# B&R Automation Studio project TD52 (part 42)

#### c_anaCyclic.st - Zyklischer Code
```iecst
(*******************************************************************************
CUSTOMIZED: c_ana 		hardcoded customized analog inputs

This code is confidential and proprietary to the INNIO Company.
It may not be used in any form, or reproduced in any manner,
without written permission of the INNIO Company.
Copyright, INNIO Company, 2022

Customized modifications: -
------------------------

History:
-------
V3.90.0	??-??-2012  pankayrodney  	converted from LD
...
V4.01.0	13.11.2014 	zengerer		ADD AnalogIn Para.rCustAnaIn_LimLoLo[] and _HiHi[] and Alarm debug links
V4.02.0	24.06.2015 	zengerer		Cleanup, prototype entry[x] for documentation comments
V4.04.0 20-06-2016	Weitzer,		add CustAnaOut[17..50]
									add reserve controller output [41 .. 45]
V4.07.0 21.01.2019	zengerer		add some example lines in init to disable Reserve ANALOG IN Warning Signal Errors – NUMBER W1177 -
V4.07.1 09.05.2019	zengerer		add more bBlock[] example lines in init to disable Reserve ANALOG IN Warning Signal Errors W1336 - W1480
V4.11.1 31.01.2022	zengerer		new extended array ranges ONLY FOR USE WITH HMI Extension Package import!
V4.12.0 22.12.2022	zengerer		Outdated declarations removed: ParaFactoryDefault.bCustAnaIn_Set4mA[x], tUniAnaConf[x]
V4.13.0 21.09.2023	zengerer		Prepared spare analog output signal for VIS display (with unchanged scaling), constant for array declaration +check AO arrays

Instructions for use:
--------------------

AVOID HARDCODED Para.xxx VALUES!
You MAYBE want to enter SOME factory default values in the INIT section, but ONLY TO THE Para_FactoryDefault.xxx STRUCTURE!
._FactoryDefault values get read out only once at first controller startup, until the par_XX.dat files are automatically generated.
By this way the parameter values in Para.xxx would stay acessible according to XT4 parameter management process.

Outstandings:
------------

*******************************************************************************)

PROGRAM _CYCLIC

	(************************************************************)
	(*                                                          *)
	(*                   ANALOG INPUT SECTION                   *)
	(*                                                          *)
	(************************************************************)

//	(*Reserve analog input x *)									(* (CONFIGURATION EXAMPLE) *)
//	(*Reserveanalogwert x    *)									(* (KONFIGURATIONSBEISPIEL)*)
//	(*************************)
//	rReplaceMeWithLocaleVarName	:= IN_CU.tCustAnaIn[x].Ai;		(*edit according to project needs*) 														(*eigene Variable für Kundenanpassung hier anbinden*)
//	OUT_CU.rCustAnaIn[x] ;										(*Use this value for plant specific extensions in other metamodules (needs .vvm edit)*)		(*OUT- Modulschnittstelle zur möglichen Verwendung in anderer Module (.vvm editieren)*)
//
//	(*scaling parameter watch*)									(*scaling parameter are used in HAL only IF NO EPLAN SCALING DATA IS PROVIDED!	*)
//	Para.rCustAnaIn_ScalMin[x]	; 	MM2VIS.bMsg1177;			(* statement here is for watch info only. AVOID HARDCODED PARA VALUES *)
//	Para.rCustAnaIn_ScalMax[x]	;								(* statement here is for watch info only. AVOID HARDCODED PARA VALUES *)
//
//	(*warning and alarm limit watch*)
//	Para.rCustAnaIn_LimLoLo[x]	;	MM2VIS.bMsg8966;			(* Alarm HiHi and LoLo, statement here is for watch info only. AVOID HARDCODED PARA VALUES *)
//	Para.rCustAnaIn_LimLo[x]	;	MM2VIS.bMsg1301;			(* Warning, statement here is for watch info only. AVOID HARDCODED PARA VALUES *)
//	Para.rCustAnaIn_LimHi[x]	; 	MM2VIS.bMsg1302;			(* Warning, statement here is for watch info only. AVOID HARDCODED PARA VALUES *)
//	Para.rCustAnaIn_LimHiHi[x]	; 								(* 						statement here is for watch info only. AVOID HARDCODED PARA VALUES *)
//	Para.rCustAnaIn_Hy[x]	; 									(* 						statement here is for watch info only. AVOID HARDCODED PARA VALUES *)
//	Para.iCustAnaIn_MinMaxActive[x];							(* see task header for settings in Para File or in INIT Para_FactoryDefault.iCustAnaIn_MinMaxActive; statement here is for watch info only. *)
//  --> see also Documents - 'CustomizedSpareRegulars' for hints on repeatedly used customisations

	(*Reserve analog input 1 *)
	(*Reserveanalogwert 1    *)
	(*************************)
	rReplaceMeWithLocaleVarName	:= IN_CU.tCustAnaIn[1].Ai;		(*edit according to project needs*)
	OUT_CU.rCustAnaIn[1] ;

	(*scaling parameter watch*)
	Para.rCustAnaIn_ScalMin[1]	; 	MM2VIS.bMsg1177;
	Para.rCustAnaIn_ScalMax[1]	;
	(*warning and alarm limit watch*)
	Para.rCustAnaIn_LimHiHi[1]	; 	MM2VIS.bMsg8966;
	Para.rCustAnaIn_LimLo[1]	;	MM2VIS.bMsg1301;
	Para.rCustAnaIn_LimHi[1]	; 	MM2VIS.bMsg1302;
	Para.rCustAnaIn_LimLoLo[1]	;	MM2VIS.bMsg8966;
	Para.rCustAnaIn_Hy[1]	;
	Para.iCustAnaIn_MinMaxActive[1];

	(*Reserve analog input 2 *)
	(*Reserveanalogwert 2    *)
	(*************************)
	rReplaceMeWithLocaleVarName	:= IN_CU.tCustAnaIn[2].Ai;
	OUT_CU.rCustAnaIn[2] ;

	(*scaling parameter watch*)
	Para.rCustAnaIn_ScalMin[2]	;	MM2VIS.bMsg1178;
	Para.rCustAnaIn_ScalMax[2]	;
	(*warning and alarm limit watch*)
	Para.rCustAnaIn_LimHiHi[2]	; 	MM2VIS.bMsg8967;
	Para.rCustAnaIn_LimLo[2]	;	MM2VIS.bMsg1304;
	Para.rCustAnaIn_LimHi[2]	; 	MM2VIS.bMsg1305;
	Para.rCustAnaIn_LimLoLo[2]	;	MM2VIS.bMsg8967;
	Para.rCustAnaIn_Hy[2]	;
	Para.iCustAnaIn_MinMaxActive[2];

	(*Reserve analog input 3 *)
	(*Reserveanalogwert 3    *)
	(*************************)
	rReplaceMeWithLocaleVarName := IN_CU.tCustAnaIn[3].Ai;
	OUT_CU.rCustAnaIn[3] ;

	Para.rCustAnaIn_ScalMin[3]	;	MM2VIS.bMsg1179;
	Para.rCustAnaIn_ScalMax[3]	;
	(*warning and alarm limit watch*)
	Para.rCustAnaIn_LimLo[3]	;	MM2VIS.bMsg1307;
	Para.rCustAnaIn_LimHi[3]	; 	MM2VIS.bMsg1308;
	Para.rCustAnaIn_LimLoLo[3]	;	MM2VIS.bMsg8968;
	Para.rCustAnaIn_LimHiHi[3]	;
	Para.rCustAnaIn_Hy[3]	;
	Para.iCustAnaIn_MinMaxActive[3];

	(*Reserve analog input 4 *)
	(*Reserveanalogwert 4    *)
	(*************************)
	rReplaceMeWithLocaleVarName := IN_CU.tCustAnaIn[4].Ai;
	OUT_CU.rCustAnaIn[4] ;

	(*scaling parameter watch*)
	Para.rCustAnaIn_ScalMin[4]	;	 MM2VIS.bMsg1180;
	Para.rCustAnaIn_ScalMax[4]	;
	(*warning and alarm limit watch*)
	Para.rCustAnaIn_LimLo[4]	;	MM2VIS.bMsg1310;
	Para.rCustAnaIn_LimHi[4]	; 	MM2VIS.bMsg1311;
	Para.rCustAnaIn_LimLoLo[4]	;	MM2VIS.bMsg8969;
	Para.rCustAnaIn_LimHiHi[4]	;
	Para.rCustAnaIn_Hy[4]	;
	Para.iCustAnaIn_MinMaxActive[4];

	(*Reserve analog input 5 *)
	(*Reserveanalogwert 5    *)
	(*************************)
	rReplaceMeWithLocaleVarName := IN_CU.tCustAnaIn[5].Ai;
	OUT_CU.rCustAnaIn[5] ;

	(*scaling parameter watch*)
	Para.rCustAnaIn_ScalMin[5]	;	 MM2VIS.bMsg1181;
	Para.rCustAnaIn_ScalMax[5]	;
	(*warning and alarm limit watch*)
	Para.rCustAnaIn_LimLo[5]	;	MM2VIS.bMsg1313;
	Para.rCustAnaIn_LimHi[5]	; 	MM2VIS.bMsg1314;
	Para.rCustAnaIn_LimLoLo[5]	;	MM2VIS.bMsg8970;
	Para.rCustAnaIn_LimHiHi[5]	;

	(*Reserveanalogwert 6 *)
	(**********************)
	rReplaceMeWithLocaleVarName := IN_CU.tCustAnaIn[6].Ai;
	OUT_CU.rCustAnaIn[6] ;

	(*scaling parameter watch*)
	Para.rCustAnaIn_ScalMin[6]	;	 MM2VIS.bMsg1182;
	Para.rCustAnaIn_ScalMax[6]	;
	(*warning and alarm limit watch*)
	Para.rCustAnaIn_LimLo[6]	;	MM2VIS.bMsg1316;
	Para.rCustAnaIn_LimHi[6]	; 	MM2VIS.bMsg1317;
	Para.rCustAnaIn_LimLoLo[6]	;	MM2VIS.bMsg8971;
	Para.rCustAnaIn_LimHiHi[6]	;

	(*Reserveanalogwert 7 *)
	(**********************)
	rReplaceMeWithLocaleVarName := IN_CU.tCustAnaIn[7].Ai;
	OUT_CU.rCustAnaIn[7] ;

	(*scaling parameter watch*)
	Para.rCustAnaIn_ScalMin[7]	;	 MM2VIS.bMsg1183;
	Para.rCustAnaIn_ScalMax[7]	;
	(*warning and alarm limit watch*)
	Para.rCustAnaIn_LimLo[7]	;	MM2VIS.bMsg1319;
	Para.rCustAnaIn_LimHi[7]	; 	MM2VIS.bMsg1320;
	Para.rCustAnaIn_LimLoLo[7]	;	MM2VIS.bMsg8972;
	Para.rCustAnaIn_LimHiHi[7]	;

	(*Reserveanalogwert 8 *)
	(**********************)
	rReplaceMeWithLocaleVarName	:= IN_CU.tCustAnaIn[8].Ai;
	OUT_CU.rCustAnaIn[8] ;

	(*scaling parameter watch*)
	Para.rCustAnaIn_ScalMin[8]	;	 MM2VIS.bMsg1184;
	Para.rCustAnaIn_ScalMax[8]	;
	(*warning and alarm limit watch*)
	Para.rCustAnaIn_LimLo[8]	;	MM2VIS.bMsg1322;
	Para.rCustAnaIn_LimHi[8]	; 	MM2VIS.bMsg1323;
	Para.rCustAnaIn_LimLoLo[8]	;	MM2VIS.bMsg8973;
	Para.rCustAnaIn_LimHiHi[8]	;

	(*Reserveanalogwert 9 *)
	(**********************)
	rReplaceMeWithLocaleVarName	:= IN_CU.tCustAnaIn[9].Ai;
	OUT_CU.rCustAnaIn[9] := 0;
	MM2VIS.bMsg1327;

	(*scaling parameter watch*)
	Para.rCustAnaIn_ScalMin[9]	;	MM2VIS.bMsg1327;	(*!change in numbering pattern!*)
	Para.rCustAnaIn_ScalMax[9]	;
	(*warning and alarm limit watch*)
	Para.rCustAnaIn_LimLo[9]	;	MM2VIS.bMsg1325;
	Para.rCustAnaIn_LimHi[9]	; 	MM2VIS.bMsg1326;
	Para.rCustAnaIn_LimLoLo[9]	;	MM2VIS.bMsg8974;
	Para.rCustAnaIn_LimHiHi[9]	;

	(*Reserveanalogwert 10 *)
	(**********************)
	rReplaceMeWithLocaleVarName	:= IN_CU.tCustAnaIn[10].Ai;
	OUT_CU.rCustAnaIn[10] := 0;
	MM2VIS.bMsg1330;

	(*scaling parameter watch*)
	Para.rCustAnaIn_ScalMin[10]	;	MM2VIS.bMsg1330;
	Para.rCustAnaIn_ScalMax[10]	;
	(*warning and alarm limit watch*)
	Para.rCustAnaIn_LimLo[10]	;	MM2VIS.bMsg1328;
	Para.rCustAnaIn_LimHi[10]	; 	MM2VIS.bMsg1329;
	Para.rCustAnaIn_LimLoLo[10]	;	MM2VIS.bMsg8975;
	Para.rCustAnaIn_LimHiHi[10]	;
	Para.rCustAnaIn_Hy[10]	;
	Para.iCustAnaIn_MinMaxActive[10];

	(*Reserveanalogwert 11 *)
	(**********************)
	rReplaceMeWithLocaleVarName	:= IN_CU.tCustAnaIn[11].Ai;
	OUT_CU.rCustAnaIn[11] := 0;
	MM2VIS.bMsg1333;

	(*scaling parameter watch*)
	Para.rCustAnaIn_ScalMin[11]	;	MM2VIS.bMsg1333;
	Para.rCustAnaIn_ScalMax[11]	;
	(*warning and alarm limit watch*)
	Para.rCustAnaIn_LimLo[11]	;	MM2VIS.bMsg1331;
	Para.rCustAnaIn_LimHi[11]	; 	MM2VIS.bMsg1332;
	Para.rCustAnaIn_LimLoLo[11]	;	MM2VIS.bMsg8976;
	Para.rCustAnaIn_LimHiHi[11]	;

	(*Reserveanalogwert 12 *)
	(**********************)
	rReplaceMeWithLocaleVarName	:= IN_CU.tCustAnaIn[12].Ai;
	OUT_CU.rCustAnaIn[12] := 0;
	MM2VIS.bMsg1336;
	(*...*)

	(*Reserveanalogwert 13 *)
	(**********************)
	rReplaceMeWithLocaleVarName	:= IN_CU.tCustAnaIn[13].Ai;
	OUT_CU.rCustAnaIn[13] := 0;
	MM2VIS.bMsg1339;

	(*Reserveanalogwert 14 *)
	(**********************)
	rReplaceMeWithLocaleVarName := IN_CU.tCustAnaIn[14].Ai;
	OUT_CU.rCustAnaIn[14] := 0;
	MM2VIS.bMsg1342;

	(*Reserveanalogwert 15 *)
	(**********************)
	rReplaceMeWithLocaleVarName	:= IN_CU.tCustAnaIn[15].Ai;
	OUT_CU.rCustAnaIn[15] := 0;
	MM2VIS.bMsg1345;

	(*Reserveanalogwert 16 *)
	(**********************)
	rReplaceMeWithLocaleVarName	:= IN_CU.tCustAnaIn[16].Ai;
	OUT_CU.rCustAnaIn[16] := 0;
	MM2VIS.bMsg1348;

	(*Reserveanalogwert 17 *)
	(**********************)
	rReplaceMeWithLocaleVarName	:= IN_CU.tCustAnaIn[17].Ai;
	OUT_CU.rCustAnaIn[17] := 0;
	MM2VIS.bMsg1351;

	(*Reserveanalogwert 18 *)
	(**********************)
	rReplaceMeWithLocaleVarName	:= IN_CU.tCustAnaIn[18].Ai;
	OUT_CU.rCustAnaIn[18] := 0;
	MM2VIS.bMsg1354;

	(*Reserveanalogwert 19 *)
	(**********************)
	rReplaceMeWithLocaleVarName	:= IN_CU.tCustAnaIn[19].Ai;
	OUT_CU.rCustAnaIn[19] := 0;
	MM2VIS.bMsg1357;

	(*Reserveanalogwert 20 *)
	(**********************)
	rReplaceMeWithLocaleVarName	:= IN_CU.tCustAnaIn[20].Ai;
	OUT_CU.rCustAnaIn[20] := 0;

	(*scaling parameter watch*)
	Para.rCustAnaIn_ScalMin[20]	;	MM2VIS.bMsg1360;
	Para.rCustAnaIn_ScalMax[20]	;
	(*warning and alarm limit watch*)
	Para.rCustAnaIn_LimLo[20]	;	MM2VIS.bMsg1358;
	Para.rCustAnaIn_LimHi[20]	; 	MM2VIS.bMsg1359;
	Para.rCustAnaIn_LimLoLo[20]	;	MM2VIS.bMsg8985;
	Para.rCustAnaIn_LimHiHi[20]	;
	Para.rCustAnaIn_Hy[20]	;
	Para.iCustAnaIn_MinMaxActive[20];

	(*Reserveanalogwert 21 *)
	(**********************)
	rReplaceMeWithLocaleVarName	:= IN_CU.tCustAnaIn[21].Ai;
	OUT_CU.rCustAnaIn[21] := 0;

	(*scaling parameter watch*)
	Para.rCustAnaIn_ScalMin[21]	;	MM2VIS.bMsg1363;
	Para.rCustAnaIn_ScalMax[21]	;
	(*warning and alarm limit watch*)
	Para.rCustAnaIn_LimLo[21]	;	MM2VIS.bMsg1361;
	Para.rCustAnaIn_LimHi[21]	; 	MM2VIS.bMsg1362;
	Para.rCustAnaIn_LimLoLo[21]	;	MM2VIS.bMsg8986;
	Para.rCustAnaIn_LimHiHi[21]	;
	Para.rCustAnaIn_Hy[21]	;
	Para.iCustAnaIn_MinMaxActive[21];

	(*Reserveanalogwert 22 *)
	(**********************)
	rReplaceMeWithLocaleVarName	:= IN_CU.tCustAnaIn[22].Ai;
	OUT_CU.rCustAnaIn[22] := 0;
	MM2VIS.bMsg1366;

	(*Reserveanalogwert 23 *)
	(**********************)
	rReplaceMeWithLocaleVarName	:= IN_CU.tCustAnaIn[23].Ai;
	OUT_CU.rCustAnaIn[23] := 0;
	MM2VIS.bMsg1369;

	(*Reserveanalogwert 24 *)
	(**********************)
	rReplaceMeWithLocaleVarName	:= IN_CU.tCustAnaIn[24].Ai;
	OUT_CU.rCustAnaIn[24] := 0;

	(*Reserveanalogwert 25 *)
	(**********************)
	rReplaceMeWithLocaleVarName	:= IN_CU.tCustAnaIn[25].Ai;
	OUT_CU.rCustAnaIn[25] := 0;

	(*Reserveanalogwert 26 *)
	(**********************)
	rReplaceMeWithLocaleVarName	:= IN_CU.tCustAnaIn[26].Ai;
	OUT_CU.rCustAnaIn[26] := 0;

	(*Reserveanalogwert 27 *)
	(**********************)
	rReplaceMeWithLocaleVarName	:= IN_CU.tCustAnaIn[27].Ai;
	OUT_CU.rCustAnaIn[27] := 0;

	(*Reserveanalogwert 28 *)
	(**********************)
	rReplaceMeWithLocaleVarName	:= IN_CU.tCustAnaIn[28].Ai;
	OUT_CU.rCustAnaIn[28] := 0;

	(*Reserveanalogwert 29 *)
	(**********************)
	rReplaceMeWithLocaleVarName	:= IN_CU.tCustAnaIn[29].Ai;
	OUT_CU.rCustAnaIn[29] := 0;

	(*Reserve analog value  30 *)
	(**************************)
	rReplaceMeWithLocaleVarName	:= IN_CU.tCustAnaIn[30].Ai;
	OUT_CU.rCustAnaIn[30] := 0;

	(*scaling parameter watch*)
	Para.rCustAnaIn_ScalMin[30]	;	MM2VIS.bMsg1390;	 	(* ANALOG IN 30 Warning Signal Error. statement here is for watch info only. *)
	Para.rCustAnaIn_ScalMax[30]	;
	(*warning and alarm limit watch*)
	Para.rCustAnaIn_LimLo[30]	;	MM2VIS.bMsg1388;
	Para.rCustAnaIn_LimHi[30]	; 	MM2VIS.bMsg1389;
	Para.rCustAnaIn_LimLoLo[30]	;	MM2VIS.bMsg8995;
	Para.rCustAnaIn_LimHiHi[30]	;
	Para.rCustAnaIn_Hy[30]	;
	Para.iCustAnaIn_MinMaxActive[30];

	(*Reserve analog value  31 *)
	(**************************)
	rReplaceMeWithLocaleVarName	:= IN_CU.tCustAnaIn[31].Ai;
	OUT_CU.rCustAnaIn[31] := 0;

	(*scaling parameter watch*)
	Para.rCustAnaIn_ScalMin[31]	;	MM2VIS.bMsg1393;		(* ANALOG IN 31 Warning Signal Error. statement here is for watch info only. *)
	Para.rCustAnaIn_ScalMax[31]	;
	(*warning limit watch*)
	Para.rCustAnaIn_LimLo[31]	;	MM2VIS.bMsg1391;  		(* ANALOG IN 31 Warning Limit LOW,  statement here is for watch info only.   *)
	Para.rCustAnaIn_LimHi[31]	; 	MM2VIS.bMsg1392;  		(* ANALOG IN 31 Warning Limit HIGH, statement here is for watch info only.   *)
(*!*)Para.rCustAnaIn_LimLoLo[31];	MM2VIS.bMsg8998;		(*!	Collective Alarm for Analog inputs 31-60:  limit alarms LoLo ! *)	(* Statement here for watch info only *)
(*!*)Para.rCustAnaIn_LimHiHi[31];	MM2VIS.bMsg8999;		(*!	Collective Alarm for Analog inputs 31-60:  limit alarms HiHi  Statement here for watch info only *)
	Para.rCustAnaIn_Hy[31]	;
	Para.iCustAnaIn_MinMaxActive[31];

	(*Reserve analog value  32 *)
	(**************************)
	rReplaceMeWithLocaleVarName	:= IN_CU.tCustAnaIn[32].Ai;
	OUT_CU.rCustAnaIn[32] := 0;

	(*scaling parameter watch*)
	Para.rCustAnaIn_ScalMin[32]	;	MM2VIS.bMsg1396;		(* ANALOG IN 32 Warning Signal Error. statement here is for watch info only. *)
	Para.rCustAnaIn_ScalMax[32]	;
	(*warning and alarm limit watch*)
	Para.rCustAnaIn_LimLo[32]	;	MM2VIS.bMsg1394;  		(* ANALOG IN 32 Warning Limit LOW,  statement here is for watch info only.   *)
	Para.rCustAnaIn_LimHi[32]	; 	MM2VIS.bMsg1395;  		(* ANALOG IN 32 Warning Limit HIGH, statement here is for watch info only.   *)
	Para.rCustAnaIn_Hy[32]	;
	Para.iCustAnaIn_MinMaxActive[32];

	(*Reserve analog value  33 *)
	(**************************)
	rReplaceMeWithLocaleVarName	:= IN_CU.tCustAnaIn[33].Ai;
	OUT_CU.rCustAnaIn[33] := 0;

	(*scaling parameter watch*)
	Para.rCustAnaIn_ScalMin[33]	;	MM2VIS.bMsg1399;
	Para.rCustAnaIn_ScalMax[33]	;
	(*warning and alarm limit watch*)
	Para.rCustAnaIn_LimLo[33]	;	MM2VIS.bMsg1397;
	Para.rCustAnaIn_LimHi[33]	; 	MM2VIS.bMsg1398;
	Para.rCustAnaIn_Hy[33]	;
	Para.iCustAnaIn_MinMaxActive[33];

	(*Reserve analog value  34 *)
	(**************************)
	rReplaceMeWithLocaleVarName	:= IN_CU.tCustAnaIn[34].Ai;
	OUT_CU.rCustAnaIn[34] := 0;

	(*scaling parameter watch*)
	Para.rCustAnaIn_ScalMin[34]	;	MM2VIS.bMsg1402;
	Para.rCustAnaIn_ScalMax[34]	;
	(*warning and alarm limit watch*)
	Para.rCustAnaIn_LimLo[34]	;	MM2VIS.bMsg1400;
	Para.rCustAnaIn_LimHi[34]	; 	MM2VIS.bMsg1401;
	Para.rCustAnaIn_Hy[34]	;
	Para.iCustAnaIn_MinMaxActive[34];

	(*Reserve analog value  35 *)
	(**************************)
	rReplaceMeWithLocaleVarName	:= IN_CU.tCustAnaIn[35].Ai;
	OUT_CU.rCustAnaIn[35] := 0;

	(*scaling parameter watch*)
	Para.rCustAnaIn_ScalMin[35]	;	MM2VIS.bMsg1405;
	Para.rCustAnaIn_ScalMax[35]	;
	(*warning and alarm limit watch*)
	Para.rCustAnaIn_LimLo[35]	;	MM2VIS.bMsg1403;
	Para.rCustAnaIn_LimHi[35]	; 	MM2VIS.bMsg1404;
	Para.rCustAnaIn_Hy[35]	;
	Para.iCustAnaIn_MinMaxActive[35];

	(*Reserve analog value  36 *)
	(**************************)
	rReplaceMeWithLocaleVarName	:= IN_CU.tCustAnaIn[36].Ai;
	OUT_CU.rCustAnaIn[36] := 0;

	(*Reserve analog value  37 *)
	(**************************)
	rReplaceMeWithLocaleVarName	:= IN_CU.tCustAnaIn[37].Ai;
	OUT_CU.rCustAnaIn[37] := 0;

	(*Reserve analog value  38 *)
	(**************************)
	rReplaceMeWithLocaleVarName	:= IN_CU.tCustAnaIn[38].Ai;
	OUT_CU.rCustAnaIn[38] := 0;

	(*Reserve analog value  39 *)
	(**************************)
	rReplaceMeWithLocaleVarName	:= IN_CU.tCustAnaIn[39].Ai;
	OUT_CU.rCustAnaIn[39] := 0;

	(*Reserve analog value  40 *)
	(**************************)
	rReplaceMeWithLocaleVarName	:= IN_CU.tCustAnaIn[40].Ai;
	OUT_CU.rCustAnaIn[40] := 0;

	(*scaling parameter watch*)
	Para.rCustAnaIn_ScalMin[40]	;	MM2VIS.bMsg1420;		(* ANALOG IN 40 Warning Signal Error. statement here is for watch info only. *)
	Para.rCustAnaIn_ScalMax[40]	;
	(*warning and alarm limit watch*)
	Para.rCustAnaIn_LimLo[40]	;	MM2VIS.bMsg1418; 		(* ANALOG IN 40 Warning Limit LOW,  statement here is for watch info only.   *)
	Para.rCustAnaIn_LimHi[40]	; 	MM2VIS.bMsg1419; 		(* ANALOG IN 40 Warning Limit HIGH, statement here is for watch info only.   *)
	Para.rCustAnaIn_Hy[40]	;
	Para.iCustAnaIn_MinMaxActive[40];

	(*Reserve analog value  41 *)
	(**************************)
	rReplaceMeWithLocaleVarName	:= IN_CU.tCustAnaIn[41].Ai;
	OUT_CU.rCustAnaIn[41] := 0;

	(*scaling parameter watch*)
	Para.rCustAnaIn_ScalMin[41]	;	MM2VIS.bMsg1423;		(* ANALOG IN 41 Warning Signal Error. statement here is for watch info only. *)
	Para.rCustAnaIn_ScalMax[41]	;
	(*warning and alarm limit watch*)
	Para.rCustAnaIn_LimLo[41]	;	MM2VIS.bMsg1421; 		(* ANALOG IN 41 Warning Limit LOW,  statement here is for watch info only.   *)
	Para.rCustAnaIn_LimHi[41]	; 	MM2VIS.bMsg1422; 		(* ANALOG IN 41 Warning Limit HIGH, statement here is for watch info only.   *)
	Para.rCustAnaIn_Hy[41]	;
	Para.iCustAnaIn_MinMaxActive[41];

	(*Reserve analog value  42 *)
	(**************************)
	rReplaceMeWithLocaleVarName	:= IN_CU.tCustAnaIn[42].Ai;
	OUT_CU.rCustAnaIn[42] := 0;

	(*Reserve analog value  43 *)
	(**************************)
	rReplaceMeWithLocaleVarName	:= IN_CU.tCustAnaIn[43].Ai;
	OUT_CU.rCustAnaIn[43] := 0;

	(*Reserve analog value  44 *)
	(**************************)
	rReplaceMeWithLocaleVarName	:= IN_CU.tCustAnaIn[44].Ai;
	OUT_CU.rCustAnaIn[44] := 0;

	(*Reserve analog value  45 *)
	(**************************)
	rReplaceMeWithLocaleVarName	:= IN_CU.tCustAnaIn[45].Ai;
	OUT_CU.rCustAnaIn[45] := 0;

	(*Reserve analog value  46 *)
	(**************************)
	rReplaceMeWithLocaleVarName	:= IN_CU.tCustAnaIn[46].Ai;
	OUT_CU.rCustAnaIn[46] := 0;

	(*Reserve analog value  47 *)
	(**************************)
	rReplaceMeWithLocaleVarName	:= IN_CU.tCustAnaIn[47].Ai;
	OUT_CU.rCustAnaIn[47] := 0;

	(*Reserve analog value  48 *)
	(**************************)
	rReplaceMeWithLocaleVarName	:= IN_CU.tCustAnaIn[48].Ai;
	OUT_CU.rCustAnaIn[48] := 0;

	(*Reserve analog value  49 *)
	(**************************)
	rReplaceMeWithLocaleVarName	:= IN_CU.tCustAnaIn[49].Ai;
	OUT_CU.rCustAnaIn[49] := 0;

	(*Reserve analog value  50 *)
	(**************************)
	rReplaceMeWithLocaleVarName	:= IN_CU.tCustAnaIn[50].Ai;
	OUT_CU.rCustAnaIn[50] := 0;

	(*scaling parameter watch*)
	Para.rCustAnaIn_ScalMin[50]	;	MM2VIS.bMsg1450;		(* ANALOG IN 50 Warning Signal Error. statement here is for watch info only. *)
	Para.rCustAnaIn_ScalMax[50]	;
	(*warning and alarm limit watch*)
	Para.rCustAnaIn_LimLo[50]	;	MM2VIS.bMsg1448;			(* ANALOG IN 50 Warning Limit LOW,  statement here is for watch info only.   *)
	Para.rCustAnaIn_LimHi[50]	; 	MM2VIS.bMsg1449;			(* ANALOG IN 50 Warning Limit HIGH, statement here is for watch info only.   *)
	Para.rCustAnaIn_Hy[50]	;
	Para.iCustAnaIn_MinMaxActive[50];

	(*Reserve analog value  51 *)
	(**************************)
	rReplaceMeWithLocaleVarName	:= IN_CU.tCustAnaIn[51].Ai;
	OUT_CU.rCustAnaIn[51] := 0;

	(*Reserve analog value  52 *)
	(**************************)
	rReplaceMeWithLocaleVarName	:= IN_CU.tCustAnaIn[52].Ai;
	OUT_CU.rCustAnaIn[52] := 0;

	(*Reserve analog value  53 *)
	(**************************)
	rReplaceMeWithLocaleVarName	:= IN_CU.tCustAnaIn[53].Ai;
	OUT_CU.rCustAnaIn[53] := 0;

	(*Reserve analog value  54 *)
	(**************************)
	rReplaceMeWithLocaleVarName	:= IN_CU.tCustAnaIn[54].Ai;
	OUT_CU.rCustAnaIn[54] := 0;

	(*Reserve analog value  55 *)
	(**************************)
	rReplaceMeWithLocaleVarName	:= IN_CU.tCustAnaIn[55].Ai;
	OUT_CU.rCustAnaIn[55] := 0;

	(*Reserve analog value  56 *)
	(**************************)
	rReplaceMeWithLocaleVarName	:= IN_CU.tCustAnaIn[56].Ai;
	OUT_CU.rCustAnaIn[56] := 0;

	(*Reserve analog value  57 *)
	(**************************)
	rReplaceMeWithLocaleVarName	:= IN_CU.tCustAnaIn[57].Ai;
	OUT_CU.rCustAnaIn[57] := 0;

	(*Reserve analog value  58 *)
	(**************************)
	rReplaceMeWithLocaleVarName	:= IN_CU.tCustAnaIn[58].Ai;
	OUT_CU.rCustAnaIn[58] := 0;

	(*Reserve analog value  59 *)
	(**************************)
	rReplaceMeWithLocaleVarName	:= IN_CU.tCustAnaIn[59].Ai;
	OUT_CU.rCustAnaIn[59] := 0;

	(*Reserve analog value 60 *)
	(**************************)
	rReplaceMeWithLocaleVarName	:= IN_CU.tCustAnaIn[60].Ai;
	OUT_CU.rCustAnaIn[60] := 0;

	(*scaling parameter watch*)
	Para.rCustAnaIn_ScalMin[60]	;	MM2VIS.bMsg1480;		(* ANALOG IN 60 Warning Signal Error. statement here is for watch info only. *)
	Para.rCustAnaIn_ScalMax[60]	;
	(*warning and alarm limit watch*)
	Para.rCustAnaIn_LimLo[60]	;MM2VIS.bMsg1478 ;			(* ANALOG IN 60 Warning Limit LOW,  statement here is for watch info only.   *)
	Para.rCustAnaIn_LimHi[60]	;MM2VIS.bMsg1479 ;			(* ANALOG IN 60 Warning Limit HIGH, statement here is for watch info only.   *)
	Para.rCustAnaIn_Hy[60]	;
	Para.iCustAnaIn_MinMaxActive[60];

	(********************************************************************************************************************************************)
	(* Reserve analog input 61 and above are not prepared in HMI default! - FOR USE ONLY WITH `HMI_Extension` Package! *)
	(* Analog inputs 61- and above have no alarm messages and HMI display prepared in default and need HMI_Update packets imported for function! *)
	(*********************************************************************************************************************************************)
	(*Reserve analog value  61 *)
	(**************************)
	rReplaceMeWithLocaleVarName	:= IN_CU.tCustAnaIn[61].Ai;
	OUT_CU.rCustAnaIn[61] := 0;

	(*Reserve analog value  62 *)
	(**************************)
	rReplaceMeWithLocaleVarName	:= IN_CU.tCustAnaIn[62].Ai;
	OUT_CU.rCustAnaIn[62] := 0;

	(*Reserve analog value  63 *)
	(**************************)
	rReplaceMeWithLocaleVarName	:= IN_CU.tCustAnaIn[63].Ai;
	OUT_CU.rCustAnaIn[63] := 0;

	(*Reserve analog value  64 *)
	(**************************)
	rReplaceMeWithLocaleVarName	:= IN_CU.tCustAnaIn[64].Ai;
	OUT_CU.rCustAnaIn[64] := 0;

	(*Reserve analog value  66 *)
	(**************************)
	rReplaceMeWithLocaleVarName	:= IN_CU.tCustAnaIn[65].Ai;
	OUT_CU.rCustAnaIn[65] := 0;

	(*Reserve analog value  66 *)
	(**************************)
	rReplaceMeWithLocaleVarName	:= IN_CU.tCustAnaIn[66].Ai;
	OUT_CU.rCustAnaIn[66] := 0;

	(*Reserve analog value  67 *)
	(**************************)
	rReplaceMeWithLocaleVarName	:= IN_CU.tCustAnaIn[67].Ai;
	OUT_CU.rCustAnaIn[67] := 0;

	(*Reserve analog value  68 *)
	(**************************)
	rReplaceMeWithLocaleVarName	:= IN_CU.tCustAnaIn[68].Ai;
	OUT_CU.rCustAnaIn[68] := 0;

	(*Reserve analog value  69 *)
	(**************************)
	rReplaceMeWithLocaleVarName	:= IN_CU.tCustAnaIn[69].Ai;
	OUT_CU.rCustAnaIn[69] := 0;

	(*Reserve analog value 70 *)
	(**************************)
	rReplaceMeWithLocaleVarName	:= IN_CU.tCustAnaIn[70].Ai;
	OUT_CU.rCustAnaIn[70] := 0;

	(*scaling parameter watch*)
	Para.rCustAnaIn_ScalMin[70]	;	MM2VIS.bMsg3810;		(* ANALOG IN 70 Warning Signal Error. statement here is for watch info only. *)
	Para.rCustAnaIn_ScalMax[70]	;
	(*warning and alarm limit watch*)
	Para.rCustAnaIn_LimLo[70]	;MM2VIS.bMsg3808 ;			(* ANALOG IN 70 Warning Limit LOW,  statement here is for watch info only.   *)
	Para.rCustAnaIn_LimHi[70]	;MM2VIS.bMsg3809 ;			(* ANALOG IN 70 Warning Limit HIGH, statement here is for watch info only.   *)
	Para.rCustAnaIn_Hy[70]	;
	Para.iCustAnaIn_MinMaxActive[70];

	(*Reserve analog value  71 *)
	(**************************)
	rReplaceMeWithLocaleVarName	:= IN_CU.tCustAnaIn[71].Ai;
	OUT_CU.rCustAnaIn[71] := 0;

	(*Reserve analog value  72 *)
	(**************************)
	rReplaceMeWithLocaleVarName	:= IN_CU.tCustAnaIn[72].Ai;
	OUT_CU.rCustAnaIn[72] := 0;

	(*Reserve analog value  73 *)
	(**************************)
	rReplaceMeWithLocaleVarName	:= IN_CU.tCustAnaIn[73].Ai;
	OUT_CU.rCustAnaIn[73] := 0;

	(*Reserve analog value  74 *)
	(**************************)
	rReplaceMeWithLocaleVarName	:= IN_CU.tCustAnaIn[74].Ai;
	OUT_CU.rCustAnaIn[74] := 0;

	(*Reserve analog value  75 *)
	(**************************)
	rReplaceMeWithLocaleVarName	:= IN_CU.tCustAnaIn[75].Ai;
	OUT_CU.rCustAnaIn[75] := 0;

	(*Reserve analog value  76 *)
	(**************************)
	rReplaceMeWithLocaleVarName	:= IN_CU.tCustAnaIn[76].Ai;
	OUT_CU.rCustAnaIn[76] := 0;

	(*Reserve analog value  77 *)
	(**************************)
	rReplaceMeWithLocaleVarName	:= IN_CU.tCustAnaIn[77].Ai;
	OUT_CU.rCustAnaIn[77] := 0;

	(*Reserve analog value  78 *)
	(**************************)
	rReplaceMeWithLocaleVarName	:= IN_CU.tCustAnaIn[78].Ai;
	OUT_CU.rCustAnaIn[78] := 0;

	(*Reserve analog value  79 *)
	(**************************)
	rReplaceMeWithLocaleVarName	:= IN_CU.tCustAnaIn[79].Ai;
	OUT_CU.rCustAnaIn[79] := 0;

	(*Reserve analog value 80 *)
	(**************************)
	rReplaceMeWithLocaleVarName	:= IN_CU.tCustAnaIn[80].Ai;
	OUT_CU.rCustAnaIn[80] := 0;

	(*scaling parameter watch*)
	Para.rCustAnaIn_ScalMin[80]	;	MM2VIS.bMsg3840;		(* ANALOG IN 80 Warning Signal Error. statement here is for watch info only. *)
	Para.rCustAnaIn_ScalMax[80]	;
	(*warning and alarm limit watch*)
	Para.rCustAnaIn_LimLo[80]	;MM2VIS.bMsg3838 ;			(* ANALOG IN 80 Warning Limit LOW,  statement here is for watch info only.   *)
	Para.rCustAnaIn_LimHi[80]	;MM2VIS.bMsg3839 ;			(* ANALOG IN 80 Warning Limit HIGH, statement here is for watch info only.   *)
	Para.rCustAnaIn_Hy[80]	;
	Para.iCustAnaIn_MinMaxActive[80];

	(*Reserve analog value  81 *)
	(**************************)
	rReplaceMeWithLocaleVarName	:= IN_CU.tCustAnaIn[81].Ai;
	OUT_CU.rCustAnaIn[81] := 0;

	(*Reserve analog value  82 *)
	(**************************)
	rReplaceMeWithLocaleVarName	:= IN_CU.tCustAnaIn[82].Ai;
	OUT_CU.rCustAnaIn[82] := 0;

	(*Reserve analog value  83 *)
	(**************************)
	rReplaceMeWithLocaleVarName	:= IN_CU.tCustAnaIn[83].Ai;
	OUT_CU.rCustAnaIn[83] := 0;

	(*Reserve analog value  84 *)
	(**************************)
	rReplaceMeWithLocaleVarName	:= IN_CU.tCustAnaIn[84].Ai;
	OUT_CU.rCustAnaIn[84] := 0;

	(*Reserve analog value  85 *)
	(**************************)
	rReplaceMeWithLocaleVarName	:= IN_CU.tCustAnaIn[85].Ai;
	OUT_CU.rCustAnaIn[85] := 0;

	(*Reserve analog value  86 *)
	(**************************)
	rReplaceMeWithLocaleVarName	:= IN_CU.tCustAnaIn[86].Ai;
	OUT_CU.rCustAnaIn[86] := 0;

	(*Reserve analog value  87 *)
	(**************************)
	rReplaceMeWithLocaleVarName	:= IN_CU.tCustAnaIn[87].Ai;
	OUT_CU.rCustAnaIn[87] := 0;

	(*Reserve analog value  88 *)
	(**************************)
	rReplaceMeWithLocaleVarName	:= IN_CU.tCustAnaIn[88].Ai;
	OUT_CU.rCustAnaIn[88] := 0;

	(*Reserve analog value  89 *)
	(**************************)
	rReplaceMeWithLocaleVarName	:= IN_CU.tCustAnaIn[89].Ai;
	OUT_CU.rCustAnaIn[89] := 0;

	(*Reserve analog value 90 *)
	(**************************)
	rReplaceMeWithLocaleVarName	:= IN_CU.tCustAnaIn[90].Ai;
	OUT_CU.rCustAnaIn[90] := 0;

	(*scaling parameter watch*)
	Para.rCustAnaIn_ScalMin[90]	;	MM2VIS.bMsg3870;		(* ANALOG IN 90 Warning Signal Error. statement here is for watch info only. *)
	Para.rCustAnaIn_ScalMax[90]	;
	(*warning and alarm limit watch*)
	Para.rCustAnaIn_LimLo[90]	;MM2VIS.bMsg3868 ;			(* ANALOG IN 90 Warning Limit LOW,  statement here is for watch info only.   *)
	Para.rCustAnaIn_LimHi[90]	;MM2VIS.bMsg3869 ;			(* ANALOG IN 90 Warning Limit HIGH, statement here is for watch info only.   *)
	Para.rCustAnaIn_Hy[90]	;
	Para.iCustAnaIn_MinMaxActive[90];

	(*Reserve analog value  91 *)
	(**************************)
	rReplaceMeWithLocaleVarName	:= IN_CU.tCustAnaIn[91].Ai;
	OUT_CU.rCustAnaIn[91] := 0;

	(*Reserve analog value  92 *)
	(**************************)
	rReplaceMeWithLocaleVarName	:= IN_CU.tCustAnaIn[92].Ai;
	OUT_CU.rCustAnaIn[92] := 0;

	(*Reserve analog value  93 *)
	(**************************)
	rReplaceMeWithLocaleVarName	:= IN_CU.tCustAnaIn[93].Ai;
	OUT_CU.rCustAnaIn[93] := 0;

	(*Reserve analog value  94 *)
	(**************************)
	rReplaceMeWithLocaleVarName	:= IN_CU.tCustAnaIn[94].Ai;
	OUT_CU.rCustAnaIn[94] := 0;

	(*Reserve analog value  95 *)
	(**************************)
	rReplaceMeWithLocaleVarName	:= IN_CU.tCustAnaIn[95].Ai;
	OUT_CU.rCustAnaIn[95] := 0;

	(*Reserve analog value  96 *)
	(**************************)
	rReplaceMeWithLocaleVarName	:= IN_CU.tCustAnaIn[96].Ai;
	OUT_CU.rCustAnaIn[96] := 0;

	(*Reserve analog value  97 *)
	(**************************)
	rReplaceMeWithLocaleVarName	:= IN_CU.tCustAnaIn[97].Ai;
	OUT_CU.rCustAnaIn[97] := 0;

	(*Reserve analog value  98 *)
	(**************************)
	rReplaceMeWithLocaleVarName	:= IN_CU.tCustAnaIn[98].Ai;
	OUT_CU.rCustAnaIn[98] := 0;

	(*Reserve analog value  99 *)
	(**************************)
	rReplaceMeWithLocaleVarName	:= IN_CU.tCustAnaIn[99].Ai;
	OUT_CU.rCustAnaIn[99] := 0;

	(*Reserve analog value 100 *)
	(**************************)
	rReplaceMeWithLocaleVarName	:= IN_CU.tCustAnaIn[100].Ai;
	OUT_CU.rCustAnaIn[100] := 0;

	(*scaling parameter watch*)
	Para.rCustAnaIn_ScalMin[100];	MM2VIS.bMsg3900;		(* ANALOG IN 100 Warning Signal Error. statement here is for watch info only. *)
	Para.rCustAnaIn_ScalMax[100];
	(*warning and alarm limit watch*)
	Para.rCustAnaIn_LimLo[100]	;MM2VIS.bMsg3898 ;			(* ANALOG IN 100 Warning Limit LOW,  statement here is for watch info only.   *)
	Para.rCustAnaIn_LimHi[100]	;MM2VIS.bMsg3899 ;			(* ANALOG IN 100 Warning Limit HIGH, statement here is for watch info only.   *)
	Para.rCustAnaIn_Hy[100]	;
	Para.iCustAnaIn_MinMaxActive[100];

	(*Reserve analog value  101 *)
	(**************************)
	rReplaceMeWithLocaleVarName	:= IN_CU.tCustAnaIn[101].Ai;
	OUT_CU.rCustAnaIn[101] := 0;

	(*Reserve analog value  102 *)
	(**************************)
	rReplaceMeWithLocaleVarName	:= IN_CU.tCustAnaIn[102].Ai;
	OUT_CU.rCustAnaIn[102] := 0;

	(*Reserve analog value  103 *)
	(**************************)
	rReplaceMeWithLocaleVarName	:= IN_CU.tCustAnaIn[103].Ai;
	OUT_CU.rCustAnaIn[103] := 0;

	(*Reserve analog value  104 *)
	(**************************)
	rReplaceMeWithLocaleVarName	:= IN_CU.tCustAnaIn[104].Ai;
	OUT_CU.rCustAnaIn[104] := 0;

	(*Reserve analog value  105 *)
	(**************************)
	rReplaceMeWithLocaleVarName	:= IN_CU.tCustAnaIn[105].Ai;
	OUT_CU.rCustAnaIn[105] := 0;

	(*Reserve analog value  106 *)
	(**************************)
	rReplaceMeWithLocaleVarName	:= IN_CU.tCustAnaIn[106].Ai;
	OUT_CU.rCustAnaIn[106] := 0;

	(*Reserve analog value  107 *)
	(**************************)
	rReplaceMeWithLocaleVarName	:= IN_CU.tCustAnaIn[107].Ai;
	OUT_CU.rCustAnaIn[107] := 0;

	(*Reserve analog value  108 *)
	(**************************)
	rReplaceMeWithLocaleVarName	:= IN_CU.tCustAnaIn[108].Ai;
	OUT_CU.rCustAnaIn[108] := 0;

	(*Reserve analog value  109 *)
	(**************************)
	rReplaceMeWithLocaleVarName	:= IN_CU.tCustAnaIn[109].Ai;
	OUT_CU.rCustAnaIn[109] := 0;

	(*Reserve analog value 110 *)
	(**************************)
	rReplaceMeWithLocaleVarName	:= IN_CU.tCustAnaIn[110].Ai;
	OUT_CU.rCustAnaIn[110] := 0;

	(*scaling parameter watch*)
	Para.rCustAnaIn_ScalMin[110];	MM2VIS.bMsg3930;		(* ANALOG IN 110 Warning Signal Error. statement here is for watch info only. *)
	Para.rCustAnaIn_ScalMax[110];
	(*warning and alarm limit watch*)
	Para.rCustAnaIn_LimLo[110]	;MM2VIS.bMsg3928 ;			(* ANALOG IN 110 Warning Limit LOW,  statement here is for watch info only.   *)
	Para.rCustAnaIn_LimHi[110]	;MM2VIS.bMsg3929 ;			(* ANALOG IN 110 Warning Limit HIGH, statement here is for watch info only.   *)
	Para.rCustAnaIn_Hy[110]	;
	Para.iCustAnaIn_MinMaxActive[110];

	(*Reserve analog value  111 *)
	(**************************)
	rReplaceMeWithLocaleVarName	:= IN_CU.tCustAnaIn[111].Ai;
	OUT_CU.rCustAnaIn[111] := 0;

	(*Reserve analog value  112 *)
	(**************************)
	rReplaceMeWithLocaleVarName	:= IN_CU.tCustAnaIn[112].Ai;
	OUT_CU.rCustAnaIn[112] := 0;

	(*Reserve analog value  113 *)
	(**************************)
	rReplaceMeWithLocaleVarName	:= IN_CU.tCustAnaIn[113].Ai;
	OUT_CU.rCustAnaIn[113] := 0;

	(*Reserve analog value  114 *)
	(**************************)
	rReplaceMeWithLocaleVarName	:= IN_CU.tCustAnaIn[114].Ai;
	OUT_CU.rCustAnaIn[114] := 0;

	(*Reserve analog value  115 *)
	(**************************)
	rReplaceMeWithLocaleVarName	:= IN_CU.tCustAnaIn[115].Ai;
	OUT_CU.rCustAnaIn[115] := 0;

	(*Reserve analog value  116 *)
	(**************************)
	rReplaceMeWithLocaleVarName	:= IN_CU.tCustAnaIn[116].Ai;
	OUT_CU.rCustAnaIn[116] := 0;

	(*Reserve analog value  117 *)
	(**************************)
	rReplaceMeWithLocaleVarName	:= IN_CU.tCustAnaIn[117].Ai;
	OUT_CU.rCustAnaIn[117] := 0;

	(*Reserve analog value  118 *)
	(**************************)
	rReplaceMeWithLocaleVarName	:= IN_CU.tCustAnaIn[118].Ai;
	OUT_CU.rCustAnaIn[118] := 0;

	(*Reserve analog value  119 *)
	(**************************)
	rReplaceMeWithLocaleVarName	:= IN_CU.tCustAnaIn[119].Ai;
	OUT_CU.rCustAnaIn[119] := 0;

	(*Reserve analog value 120 *)
	(**************************)
	rReplaceMeWithLocaleVarName	:= IN_CU.tCustAnaIn[120].Ai;
	OUT_CU.rCustAnaIn[120] := 0;

	(*scaling parameter watch*)
	Para.rCustAnaIn_ScalMin[120];	MM2VIS.bMsg3960;		(* ANALOG IN 120 Warning Signal Error. statement here is for watch info only. *)
	Para.rCustAnaIn_ScalMax[120];
	(*warning and alarm limit watch*)
	Para.rCustAnaIn_LimLo[120];		MM2VIS.bMsg3958 ;			(* ANALOG IN 120 Warning Limit LOW,  statement here is for watch info only.   *)
	Para.rCustAnaIn_LimHi[120];		MM2VIS.bMsg3959 ;			(* ANALOG IN 120 Warning Limit HIGH, statement here is for watch info only.   *)
	Para.rCustAnaIn_Hy[120];
	Para.iCustAnaIn_MinMaxActive[120];

	(*********************************************************************************************************************************)

	(*********************************************************************************************************************************)

	(********************************************************)
	(*                                                      *)
	(*                 ANALOG OUTPUT SECTION                *)
	(*                                                      *)
	(********************************************************)

//	(***************************)
//	(* Reserve analog output x *)								(* (CONFIGURATION EXAMPLE) *)
//	(* Reserveanalogausgang x  *)								(* (KONFIGURATIONSBEISPIEL)*)
//	(***************************)
//	OUT_CU.tCustAnaOut[x].Ao	:= rConnectYourVariableHere ;	(*eigene Variable für Kundenanpassung hier anbeinden*)	(*edit according to project needs*)
//
//	(*scaling parameter watch*)									(* scaling parameter are used in HAL only IF NO EPLAN SCALING DATA IS PROVIDED!	*)
//	Para.rCustAnaOut_ScalMin[x]	; 								(*[Customer Unit] 'software side' of scaling;	statement here is for watch info only. AVOID HARDCODED PARA VALUES *)
//	Para.rCustAnaOut_ScalMax[x]	;								(*[Customer Unit] 'software side' of scaling;	statement here is for watch info only. AVOID HARDCODED PARA VALUES *)
//	Para.rI_CustAnaOut_ScalMin[x] ; 	(* := 4; *)				(*[mA] 'hardware side' of scaling;				statement here is for watch info only. AVOID HARDCODED PARA VALUES *)
//	Para.rI_CustAnaOut_ScalMin[x] ;		(* := 20; *)			(*[mA] 'hardware side' of scaling;				statement here is for watch info only. AVOID HARDCODED PARA VALUES *)

	(* reserve analog output 1 *)
	OUT_CU.tCustAnaOut[1].Ao	:= rConnectYourVariableHere ;	(* change customized *)
	(*scaling parameter watch*)
	Para.rCustAnaOut_ScalMin[1]	;
	Para.rCustAnaOut_ScalMax[1]	;
	Para.rI_CustAnaOut_ScalMin[1] ;
	Para.rI_CustAnaOut_ScalMax[1] ;
	MM2VIS.rCustAnaOut[1] ; 								(*Example call of prepared spare analog output for VIS service display; OLD: MM2VIS.rCustAnaOut_Norm[1]  *)

	(* reserve analog output 2 *)
	OUT_CU.tCustAnaOut[2].Ao	:= rConnectYourVariableHere ;
	(*scaling parameter watch*)
	Para.rCustAnaOut_ScalMin[2]	;
	Para.rCustAnaOut_ScalMax[2]	;
	Para.rI_CustAnaOut_ScalMin[2] ;
	Para.rI_CustAnaOut_ScalMax[2] ;

	(* reserve analog output 3 *)
	OUT_CU.tCustAnaOut[3].Ao	:= rConnectYourVariableHere ;
	(*scaling parameter watch*)
	Para.rCustAnaOut_ScalMin[3]	;
	Para.rCustAnaOut_ScalMax[3]	;
	Para.rI_CustAnaOut_ScalMin[3] ;
	Para.rI_CustAnaOut_ScalMax[3] ;

	(* reserve analog output 4 *)
	OUT_CU.tCustAnaOut[4].Ao	:= rConnectYourVariableHere ;
	(*scaling parameter watch*)
	Para.rCustAnaOut_ScalMin[4]	;
	Para.rCustAnaOut_ScalMax[4]	;
	Para.rI_CustAnaOut_ScalMin[4] ;
	Para.rI_CustAnaOut_ScalMax[4] ;

	(* reserve analog output 5 *)
//	OUT_CU.tCustAnaOut[5].Ao	:= rConnectYourVariableHere ;	 	(*VSofti*)
	(*scaling parameter watch*)
	Para.rCustAnaOut_ScalMin[5]	;
	Para.rCustAnaOut_ScalMax[5]	;
	Para.rI_CustAnaOut_ScalMin[5] ;
	Para.rI_CustAnaOut_ScalMax[5] ;

	(* reserve analog output 6 *)
	OUT_CU.tCustAnaOut[6].Ao	:= rConnectYourVariableHere ;
	(*scaling parameter watch*)
	Para.rCustAnaOut_ScalMin[6]	;
	Para.rCustAnaOut_ScalMax[6]	;
	Para.rI_CustAnaOut_ScalMin[6] ;
	Para.rI_CustAnaOut_ScalMax[6] ;

	(* reserve analog output 7 *)
//	OUT_CU.tCustAnaOut[7].Ao	:= rConnectYourVariableHere ;	 	(*VSofti*)
	(*scaling parameter watch*)
	Para.rCustAnaOut_ScalMin[7]	;
	Para.rCustAnaOut_ScalMax[7]	;
	Para.rI_CustAnaOut_ScalMin[7] ;
	Para.rI_CustAnaOut_ScalMax[7] ;

	(* reserve analog output 8 *)
//	OUT_CU.tCustAnaOut[8].Ao	:= rConnectYourVariableHere ;	 	(*VSofti*)
	(*scaling parameter watch*)
	Para.rCustAnaOut_ScalMin[8]	;
	Para.rCustAnaOut_ScalMax[8]	;
	Para.rI_CustAnaOut_ScalMin[8] ;
	Para.rI_CustAnaOut_ScalMax[8] ;

	(* reserve analog output 9 *)
//	OUT_CU.tCustAnaOut[9].Ao	:= rConnectYourVariableHere ;	 	(*VSofti*)
	(*scaling parameter watch*)
	Para.rCustAnaOut_ScalMin[9]	;
	Para.rCustAnaOut_ScalMax[9]	;
	Para.rI_CustAnaOut_ScalMin[9] ;
	Para.rI_CustAnaOut_ScalMax[9] ;

	(* reserve analog output 10 *)
//	OUT_CU.tCustAnaOut[10].Ao	:= rConnectYourVariableHere ;	 	(*VSofti*)
	(*scaling parameter watch*)
	Para.rCustAnaOut_ScalMin[10] ;
	Para.rCustAnaOut_ScalMax[10] ;
	Para.rI_CustAnaOut_ScalMin[10] ;
	Para.rI_CustAnaOut_ScalMax[10] ;

	(* reserve analog output 11 *)
//	OUT_CU.tCustAnaOut[11].Ao	:= rConnectYourVariableHere ;	 	(*VSofti*)
	(*scaling parameter watch*)
	Para.rCustAnaOut_ScalMin[11] ;
	Para.rCustAnaOut_ScalMax[11] ;
	Para.rI_CustAnaOut_ScalMin[11] ;
	Para.rI_CustAnaOut_ScalMax[11] ;

	(* reserve analog output 12 *)
//	OUT_CU.tCustAnaOut[12].Ao	:= rConnectYourVariableHere ;	 	(*VSofti*)
	(*scaling parameter watch*)
	Para.rCustAnaOut_ScalMin[12] ;
	Para.rCustAnaOut_ScalMax[12] ;
	Para.rI_CustAnaOut_ScalMin[12] ;
	Para.rI_CustAnaOut_ScalMax[12] ;

	(* reserve analog output 13 *)
//	OUT_CU.tCustAnaOut[13].Ao	:= rConnectYourVariableHere ;	 	(*VSofti*)
	(*scaling parameter watch*)
	Para.rCustAnaOut_ScalMin[13] ;
	Para.rCustAnaOut_ScalMax[13] ;
	Para.rI_CustAnaOut_ScalMin[13] ;
	Para.rI_CustAnaOut_ScalMax[13] ;

	(* reserve analog output 14 *)
//	OUT_CU.tCustAnaOut[14].Ao	:= rConnectYourVariableHere ;	 	(*VSofti*)
	(*scaling parameter watch*)
	Para.rCustAnaOut_ScalMin[14] ;
	Para.rCustAnaOut_ScalMax[14] ;
	Para.rI_CustAnaOut_ScalMin[14] ;
	Para.rI_CustAnaOut_ScalMax[14] ;

	(* reserve analog output 15 *)
	OUT_CU.tCustAnaOut[15].Ao	:= rConnectYourVariableHere ;
	(*scaling parameter watch*)
	Para.rCustAnaOut_ScalMin[15] ;
	Para.rCustAnaOut_ScalMax[15] ;
	Para.rI_CustAnaOut_ScalMin[15] ;
	Para.rI_CustAnaOut_ScalMax[15] ;

	(* reserve analog output 16 *)
	OUT_CU.tCustAnaOut[16].Ao	:= rConnectYourVariableHere ;
	(*scaling parameter watch*)
	Para.rCustAnaOut_ScalMin[16]	;
	Para.rCustAnaOut_ScalMax[16]	;
	Para.rI_CustAnaOut_ScalMin[16] ;
	Para.rI_CustAnaOut_ScalMax[16] ;

	(********************************************************************************************************************************************)
	(* Reserve analog output 17 and above are not prepared in HMI default! - FOR USE ONLY WITH `HMI_Extension` Package! *)
	(* Analog outputs 17- and above have no parameter values prepared in HMI display default and need HMI_Update packets imported for function! *)
	(*********************************************************************************************************************************************)

	(* reserve analog output 17 *)
	OUT_CU.tCustAnaOut[17].Ao	:= rConnectYourVariableHere ;
	(*scaling parameter watch*)
	Para.rCustAnaOut_ScalMin[17]	;
	Para.rCustAnaOut_ScalMax[17]	;
	Para.rI_CustAnaOut_ScalMin[17] ;
	Para.rI_CustAnaOut_ScalMax[17] ;

	(* reserve analog output 18 *)
	OUT_CU.tCustAnaOut[18].Ao	:= rConnectYourVariableHere ;
	(*scaling parameter watch*)
	Para.rCustAnaOut_ScalMin[18]	;
	Para.rCustAnaOut_ScalMax[18]	;
	Para.rI_CustAnaOut_ScalMin[18] ;
	Para.rI_CustAnaOut_ScalMax[18] ;

	(* reserve analog output 19 *)
	OUT_CU.tCustAnaOut[19].Ao	:= rConnectYourVariableHere ;
	(*scaling parameter watch*)
	Para.rCustAnaOut_ScalMin[19]	;
	Para.rCustAnaOut_ScalMax[19]	;
	Para.rI_CustAnaOut_ScalMin[19] ;
	Para.rI_CustAnaOut_ScalMax[19] ;

	(* reserve analog output 20 *)
	OUT_CU.tCustAnaOut[20].Ao	:= rConnectYourVariableHere ;
	(*scaling parameter watch*)
	Para.rCustAnaOut_ScalMin[20]	;
	Para.rCustAnaOut_ScalMax[20]	;
	Para.rI_CustAnaOut_ScalMin[20] ;
	Para.rI_CustAnaOut_ScalMax[20] ;

	(* reserve analog output 21 *)
	OUT_CU.tCustAnaOut[21].Ao	:= rConnectYourVariableHere ;
	(*scaling parameter watch*)
	Para.rCustAnaOut_ScalMin[21]	;
	Para.rCustAnaOut_ScalMax[21]	;
	Para.rI_CustAnaOut_ScalMin[21] ;
	Para.rI_CustAnaOut_ScalMax[21] ;

	(* reserve analog output 22 *)
	OUT_CU.tCustAnaOut[22].Ao	:= rConnectYourVariableHere ;
	(*scaling parameter watch*)
	Para.rCustAnaOut_ScalMin[22]	;
	Para.rCustAnaOut_ScalMax[22]	;
	Para.rI_CustAnaOut_ScalMin[22] ;
	Para.rI_CustAnaOut_ScalMax[22] ;

	(* reserve analog output 23 *)
	OUT_CU.tCustAnaOut[23].Ao	:= rConnectYourVariableHere ;
	(*scaling parameter watch*)
	Para.rCustAnaOut_ScalMin[23]	;
	Para.rCustAnaOut_ScalMax[23]	;
	Para.rI_CustAnaOut_ScalMin[23] ;
	Para.rI_CustAnaOut_ScalMax[23] ;

	(* reserve analog output 24 *)
	OUT_CU.tCustAnaOut[24].Ao	:= rConnectYourVariableHere ;
	(*scaling parameter watch*)
	Para.rCustAnaOut_ScalMin[24]	;
	Para.rCustAnaOut_ScalMax[24]	;
	Para.rI_CustAnaOut_ScalMin[24] ;
	Para.rI_CustAnaOut_ScalMax[24] ;

	(* reserve analog output 25 *)
	OUT_CU.tCustAnaOut[25].Ao	:= rConnectYourVariableHere ;
	(*scaling parameter watch*)
	Para.rCustAnaOut_ScalMin[25]	;
	Para.rCustAnaOut_ScalMax[25]	;
	Para.rI_CustAnaOut_ScalMin[25] ;
	Para.rI_CustAnaOut_ScalMax[25] ;

	(* reserve analog output 26 *)
	OUT_CU.tCustAnaOut[26].Ao	:= rConnectYourVariableHere ;
	(*scaling parameter watch*)
	Para.rCustAnaOut_ScalMin[26]	;
	Para.rCustAnaOut_ScalMax[26]	;
	Para.rI_CustAnaOut_ScalMin[26] ;
	Para.rI_CustAnaOut_ScalMax[26] ;

	(* reserve analog output 27 *)
	OUT_CU.tCustAnaOut[27].Ao	:= rConnectYourVariableHere ;
	(*scaling parameter watch*)
	Para.rCustAnaOut_ScalMin[27]	;
	Para.rCustAnaOut_ScalMax[27]	;
	Para.rI_CustAnaOut_ScalMin[27] ;
	Para.rI_CustAnaOut_ScalMax[27] ;

	(* reserve analog output 28 *)
	OUT_CU.tCustAnaOut[28].Ao	:= rConnectYourVariableHere ;
	(*scaling parameter watch*)
	Para.rCustAnaOut_ScalMin[28]	;
	Para.rCustAnaOut_ScalMax[28]	;
	Para.rI_CustAnaOut_ScalMin[28] ;
	Para.rI_CustAnaOut_ScalMax[28] ;

	(* reserve analog output 29 *)
	OUT_CU.tCustAnaOut[29].Ao	:= rConnectYourVariableHere ;
	(*scaling parameter watch*)
	Para.rCustAnaOut_ScalMin[29]	;
	Para.rCustAnaOut_ScalMax[29]	;
	Para.rI_CustAnaOut_ScalMin[29] ;
	Para.rI_CustAnaOut_ScalMax[29] ;

	(* reserve analog output 30 *)
	OUT_CU.tCustAnaOut[30].Ao	:= rConnectYourVariableHere ;
	(*scaling parameter watch*)
	Para.rCustAnaOut_ScalMin[30]	;
	Para.rCustAnaOut_ScalMax[30]	;
	Para.rI_CustAnaOut_ScalMin[30] ;
	Para.rI_CustAnaOut_ScalMax[30] ;

	(* reserve analog output 31 *)
	OUT_CU.tCustAnaOut[31].Ao	:= rConnectYourVariableHere ;
	(*scaling parameter watch*)
	Para.rCustAnaOut_ScalMin[31]	;
	Para.rCustAnaOut_ScalMax[31]	;
	Para.rI_CustAnaOut_ScalMin[31] ;
	Para.rI_CustAnaOut_ScalMax[31] ;

	(* reserve analog output 32 *)
	OUT_CU.tCustAnaOut[32].Ao	:= rConnectYourVariableHere ;
	(*scaling parameter watch*)
	Para.rCustAnaOut_ScalMin[32]	;
	Para.rCustAnaOut_ScalMax[32]	;
	Para.rI_CustAnaOut_ScalMin[32] ;
	Para.rI_CustAnaOut_ScalMax[32] ;

	(* reserve analog output 33 *)
	OUT_CU.tCustAnaOut[33].Ao	:= rConnectYourVariableHere ;
	(*scaling parameter watch*)
	Para.rCustAnaOut_ScalMin[33]	;
	Para.rCustAnaOut_ScalMax[33]	;
	Para.rI_CustAnaOut_ScalMin[33] ;
	Para.rI_CustAnaOut_ScalMax[33] ;

	(* reserve analog output 34 *)
	OUT_CU.tCustAnaOut[34].Ao	:= rConnectYourVariableHere ;
	(*scaling parameter watch*)
	Para.rCustAnaOut_ScalMin[34]	;
	Para.rCustAnaOut_ScalMax[34]	;
	Para.rI_CustAnaOut_ScalMin[34] ;
	Para.rI_CustAnaOut_ScalMax[34] ;

	(* reserve analog output 35 *)
	OUT_CU.tCustAnaOut[35].Ao	:= rConnectYourVariableHere ;
	(*scaling parameter watch*)
	Para.rCustAnaOut_ScalMin[35]	;
	Para.rCustAnaOut_ScalMax[35]	;
	Para.rI_CustAnaOut_ScalMin[35] ;
	Para.rI_CustAnaOut_ScalMax[35] ;

	(* reserve analog output 36 *)
	OUT_CU.tCustAnaOut[36].Ao	:= rConnectYourVariableHere ;
	(*scaling parameter watch*)
	Para.rCustAnaOut_ScalMin[36]	;
	Para.rCustAnaOut_ScalMax[36]	;
	Para.rI_CustAnaOut_ScalMin[36] ;
	Para.rI_CustAnaOut_ScalMax[36] ;

	(* reserve analog output 37 *)
	OUT_CU.tCustAnaOut[37].Ao	:= rConnectYourVariableHere ;
	(*scaling parameter watch*)
	Para.rCustAnaOut_ScalMin[37]	;
	Para.rCustAnaOut_ScalMax[37]	;
	Para.rI_CustAnaOut_ScalMin[37] ;
	Para.rI_CustAnaOut_ScalMax[37] ;

	(* reserve analog output 38 *)
	OUT_CU.tCustAnaOut[38].Ao	:= rConnectYourVariableHere ;
	(*scaling parameter watch*)
	Para.rCustAnaOut_ScalMin[38]	;
	Para.rCustAnaOut_ScalMax[38]	;
	Para.rI_CustAnaOut_ScalMin[38] ;
	Para.rI_CustAnaOut_ScalMax[38] ;

	(* reserve analog output 39 *)
	OUT_CU.tCustAnaOut[39].Ao	:= rConnectYourVariableHere ;
	(*scaling parameter watch*)
	Para.rCustAnaOut_ScalMin[39]	;
	Para.rCustAnaOut_ScalMax[39]	;
	Para.rI_CustAnaOut_ScalMin[39] ;
	Para.rI_CustAnaOut_ScalMax[39] ;

	(* reserve analog output 40 *)
	OUT_CU.tCustAnaOut[40].Ao	:= rConnectYourVariableHere ;
	(*scaling parameter watch*)
	Para.rCustAnaOut_ScalMin[40]	;
	Para.rCustAnaOut_ScalMax[40]	;
	Para.rI_CustAnaOut_ScalMin[40] ;
	Para.rI_CustAnaOut_ScalMax[40] ;

	(* reserve analog output 41 *)
	OUT_CU.tCustAnaOut[41].Ao	:= rConnectYourVariableHere ;
	(*scaling parameter watch*)
	Para.rCustAnaOut_ScalMin[41]	;
	Para.rCustAnaOut_ScalMax[41]	;
	Para.rI_CustAnaOut_ScalMin[41] ;
	Para.rI_CustAnaOut_ScalMax[41] ;

	(* reserve analog output 42 *)
	OUT_CU.tCustAnaOut[42].Ao	:= rConnectYourVariableHere ;
	(*scaling parameter watch*)
	Para.rCustAnaOut_ScalMin[42]	;
	Para.rCustAnaOut_ScalMax[42]	;
	Para.rI_CustAnaOut_ScalMin[42] ;
	Para.rI_CustAnaOut_ScalMax[42] ;

	(* reserve analog output 43 *)
	OUT_CU.tCustAnaOut[43].Ao	:= rConnectYourVariableHere ;
	(*scaling parameter watch*)
	Para.rCustAnaOut_ScalMin[43]	;
	Para.rCustAnaOut_ScalMax[43]	;
	Para.rI_CustAnaOut_ScalMin[43] ;
	Para.rI_CustAnaOut_ScalMax[43] ;

	(* reserve analog output 44 *)
	OUT_CU.tCustAnaOut[44].Ao	:= rConnectYourVariableHere ;
	(*scaling parameter watch*)
	Para.rCustAnaOut_ScalMin[44]	;
	Para.rCustAnaOut_ScalMax[44]	;
	Para.rI_CustAnaOut_ScalMin[44] ;
	Para.rI_CustAnaOut_ScalMax[44] ;

	(* reserve analog output 45 *)
	OUT_CU.tCustAnaOut[45].Ao	:= rConnectYourVariableHere ;
	(*scaling parameter watch*)
	Para.rCustAnaOut_ScalMin[45]	;
	Para.rCustAnaOut_ScalMax[45]	;
	Para.rI_CustAnaOut_ScalMin[45] ;
	Para.rI_CustAnaOut_ScalMax[45] ;

	(* reserve analog output 46 *)
	OUT_CU.tCustAnaOut[46].Ao	:= rConnectYourVariableHere ;
	(*scaling parameter watch*)
	Para.rCustAnaOut_ScalMin[46]	;
	Para.rCustAnaOut_ScalMax[46]	;
	Para.rI_CustAnaOut_ScalMin[46] ;
	Para.rI_CustAnaOut_ScalMax[46] ;

	(* reserve analog output 47 *)
	OUT_CU.tCustAnaOut[47].Ao	:= rConnectYourVariableHere ;
	(*scaling parameter watch*)
	Para.rCustAnaOut_ScalMin[47]	;
	Para.rCustAnaOut_ScalMax[47]	;
	Para.rI_CustAnaOut_ScalMin[47] ;
	Para.rI_CustAnaOut_ScalMax[47] ;

	(* reserve analog output 48 *)
	OUT_CU.tCustAnaOut[48].Ao	:= rConnectYourVariableHere ;
	(*scaling parameter watch*)
	Para.rCustAnaOut_ScalMin[48]	;
	Para.rCustAnaOut_ScalMax[48]	;
	Para.rI_CustAnaOut_ScalMin[48] ;
	Para.rI_CustAnaOut_ScalMax[48] ;

	(* reserve analog output 49 *)
	OUT_CU.tCustAnaOut[49].Ao	:= rConnectYourVariableHere ;
	(*scaling parameter watch*)
	Para.rCustAnaOut_ScalMin[49]	;
	Para.rCustAnaOut_ScalMax[49]	;
	Para.rI_CustAnaOut_ScalMin[49] ;
	Para.rI_CustAnaOut_ScalMax[49] ;

	(* reserve analog output 50 *)
	OUT_CU.tCustAnaOut[50].Ao	:= rConnectYourVariableHere ;
	(*scaling parameter watch*)
	Para.rCustAnaOut_ScalMin[50]	;
	Para.rCustAnaOut_ScalMax[50]	;
	Para.rI_CustAnaOut_ScalMin[50] ;
	Para.rI_CustAnaOut_ScalMax[50] ;

	(*********************************************************************************************************************************)
	(* Reserve analog output 51 and above prepared from V4.11 on in PLC - FOR USE ONLY WITH `HMI_Extension` Package! *)

	(* reserve analog output 51 - ONLY USE WITH HMI Extension Package import! *)
	OUT_CU.tCustAnaOut[51].Ao	:= rConnectYourVariableHere ;
	(*scaling parameter watch*)
	Para.rCustAnaOut_ScalMin[51]	;
	Para.rCustAnaOut_ScalMax[51]	;
	Para.rI_CustAnaOut_ScalMin[51]	;
	Para.rI_CustAnaOut_ScalMax[51]	;

	(* reserve analog output 52 - ONLY USE WITH HMI Extension Package import! *)
	OUT_CU.tCustAnaOut[52].Ao	:= rConnectYourVariableHere ;
	(*scaling parameter watch*)
	Para.rCustAnaOut_ScalMin[52]	;
	Para.rCustAnaOut_ScalMax[52]	;
	Para.rI_CustAnaOut_ScalMin[52]	;
	Para.rI_CustAnaOut_ScalMax[52]	;

	(* reserve analog output 53 - ONLY USE WITH HMI Extension Package import! *)
	OUT_CU.tCustAnaOut[53].Ao	:= rConnectYourVariableHere ;
	(*scaling parameter watch*)
	Para.rCustAnaOut_ScalMin[53]	;
	Para.rCustAnaOut_ScalMax[53]	;
	Para.rI_CustAnaOut_ScalMin[53]	;
	Para.rI_CustAnaOut_ScalMax[53]	;

	(* reserve analog output 54 - ONLY USE WITH HMI Extension Package import! *)
	OUT_CU.tCustAnaOut[54].Ao	:= rConnectYourVariableHere ;
	(*scaling parameter watch*)
	Para.rCustAnaOut_ScalMin[54]	;
	Para.rCustAnaOut_ScalMax[54]	;
	Para.rI_CustAnaOut_ScalMin[54]	;
	Para.rI_CustAnaOut_ScalMax[54]	;

	(* reserve analog output 55 - ONLY USE WITH HMI Extension Package import! *)
	OUT_CU.tCustAnaOut[55].Ao	:= rConnectYourVariableHere ;
	(*scaling parameter watch*)
	Para.rCustAnaOut_ScalMin[55]	;
	Para.rCustAnaOut_ScalMax[55]	;
	Para.rI_CustAnaOut_ScalMin[55]	;
	Para.rI_CustAnaOut_ScalMax[55]	;

	(* reserve analog output 56 - ONLY USE WITH HMI Extension Package import! *)
	OUT_CU.tCustAnaOut[56].Ao	:= rConnectYourVariableHere ;
	(*scaling parameter watch*)
	Para.rCustAnaOut_ScalMin[56]	;
	Para.rCustAnaOut_ScalMax[56]	;
	Para.rI_CustAnaOut_ScalMin[56]	;
	Para.rI_CustAnaOut_ScalMax[56]	;

	(* reserve analog output 57 - ONLY USE WITH HMI Extension Package import! *)
	OUT_CU.tCustAnaOut[57].Ao	:= rConnectYourVariableHere ;
	(*scaling parameter watch*)
	Para.rCustAnaOut_ScalMin[57]	;
	Para.rCustAnaOut_ScalMax[57]	;
	Para.rI_CustAnaOut_ScalMin[57]	;
	Para.rI_CustAnaOut_ScalMax[57]	;

	(* reserve analog output 58 - ONLY USE WITH HMI Extension Package import! *)
	OUT_CU.tCustAnaOut[58].Ao	:= rConnectYourVariableHere ;
	(*scaling parameter watch*)
	Para.rCustAnaOut_ScalMin[58]	;
	Para.rCustAnaOut_ScalMax[58]	;
	Para.rI_CustAnaOut_ScalMin[58]	;
	Para.rI_CustAnaOut_ScalMax[58]	;

	(* reserve analog output 59 - ONLY USE WITH HMI Extension Package import! *)
	OUT_CU.tCustAnaOut[59].Ao	:= rConnectYourVariableHere ;
	(*scaling parameter watch*)
	Para.rCustAnaOut_ScalMin[59]	;
	Para.rCustAnaOut_ScalMax[59]	;
	Para.rI_CustAnaOut_ScalMin[59]	;
	Para.rI_CustAnaOut_ScalMax[59]	;

	(* reserve analog output 60 - ONLY USE WITH HMI Extension Package import! *)
	OUT_CU.tCustAnaOut[60].Ao	:= rConnectYourVariableHere ;
	(*scaling parameter watch*)
	Para.rCustAnaOut_ScalMin[60]	;
	Para.rCustAnaOut_ScalMax[60]	;
	Para.rI_CustAnaOut_ScalMin[60]	;
	Para.rI_CustAnaOut_ScalMax[60]	;
	MM2VIS.rCustAnaOut[60] ; 								(*Example call of prepared spare analog output for VIS service display*)

	(*********************************************************************************************************************************)
	(* VIS service display values for the  prepared spare analog outputs *)
	FOR iCnt_AnaOut := 1 TO iNoOf_AnaOut DO
		MM2VIS.rCustAnaOut[iCnt_AnaOut] := OUT_CU.tCustAnaOut[iCnt_AnaOut].Ao; 		(*prepared spare analog output for VIS service display; signal scaling unchanged *)
	END_FOR
	(*********************************************************************************************************************************)

	(**********************************************************)
	(*                                                        *)
	(*                CONTROLLER OUTPUT SECTION               *)
	(*                                                        *)
	(**********************************************************)

//	(**********************************)
//	(* reserve controller output x    *)							(* (CONFIGURATION EXAMPLE)  *)
//	(* Reserveregler- Analogausgang x *)							(* (KONFIGURATIONSBEISPIEL) *)
//	(**********************************)
//	OUT_CU.tCtr_CustOut[x].Ao		:= OUT_CU.tCtr_Cust1_Out.Y;		(* most times no change necessary *)
//	(*scaling parameter watch*)
//	Para.rCtr_CustOut_ScalMin[x]	;								(* old, not used anymore *)
//	Para.rCtr_CustOut_ScalMax[x]	;								(* old, not used anymore *)
//	Para.rI_Ctr_CustOut_ScalMin[x]	;	(* := 4; *)					(*[mA]. For watch info only. AVOID HARDCODED PARA VALUES; scaling parameter are used in HAL only IF NO EPLAN SCALING DATA IS PROVIDED!	*)
//	Para.rI_Ctr_CustOut_ScalMax[x]	;	(* := 20; *)				(*[mA]. For watch info only. AVOID HARDCODED PARA VALUES; scaling parameter are used in HAL only IF NO EPLAN SCALING DATA IS PROVIDED!  *)

	(* reserve controller output 1 *)
	OUT_CU.tCtr_CustOut[1].Ao		:= OUT_CU.tCtr_Cust1_Out.Y;		(* most times no change necessary *)
	(*scaling parameter watch*)
	Para.rI_Ctr_CustOut_ScalMin[1]	;
	Para.rI_Ctr_CustOut_ScalMax[1]	;

	(* reserve controller output 2 *)
	OUT_CU.tCtr_CustOut[2].Ao		:= OUT_CU.tCtr_Cust2_Out.Y;
	(*scaling parameter watch*)
	Para.rI_Ctr_CustOut_ScalMin[2]	;
	Para.rI_Ctr_CustOut_ScalMax[2]	;

	(* reserve controller output 3 *)
	OUT_CU.tCtr_CustOut[3].Ao		:= OUT_CU.tCtr_Cust3_Out.Y;
	(*scaling parameter watch*)
	Para.rI_Ctr_CustOut_ScalMin[3]	;
	Para.rI_Ctr_CustOut_ScalMax[3]	;

	(* reserve controller output 4 *)
	OUT_CU.tCtr_CustOut[4].Ao		:= OUT_CU.tCtr_Cust4_Out.Y;
	(*scaling parameter watch*)
	Para.rI_Ctr_CustOut_ScalMin[4]	;
	Para.rI_Ctr_CustOut_ScalMax[4]	;

	(* reserve controller output 5 *)
	OUT_CU.tCtr_CustOut[5].Ao		:= OUT_CU.tCtr_Cust5_Out.Y;
	(*scaling parameter watch*)
	Para.rI_Ctr_CustOut_ScalMin[5]	;
	Para.rI_Ctr_CustOut_ScalMax[5]	;

	(* reserve controller output 6 *)
	OUT_CU.tCtr_CustOut[6].Ao		:= OUT_CU.tCtr_Cust6_Out.Y;
	(*scaling parameter watch*)
	Para.rI_Ctr_CustOut_ScalMin[6]	;
	Para.rI_Ctr_CustOut_ScalMax[6]	;

	(* reserve controller output 7 *)
	OUT_CU.tCtr_CustOut[7].Ao		:= OUT_CU.tCtr_Cust7_Out.Y;
	(*scaling parameter watch*)
	Para.rI_Ctr_CustOut_ScalMin[7]	;
	Para.rI_Ctr_CustOut_ScalMax[7]	;

	(* reserve controller output 8 *)
	OUT_CU.tCtr_CustOut[8].Ao		:= OUT_CU.tCtr_Cust8_Out.Y;
	(*scaling parameter watch*)
	Para.rI_Ctr_CustOut_ScalMin[8]	;
	Para.rI_Ctr_CustOut_ScalMax[8]	;

	(***********************************************************)

	(* reserve controller output 41 *)
	OUT_CU.tCtr_CustOut[41].Ao		:= OUT_CU.tCtr_Cust41_Out.Y;
	(*scaling parameter watch*)
	Para.rI_Ctr_CustOut_ScalMin[41]	;
	Para.rI_Ctr_CustOut_ScalMax[41]	;

	(* reserve controller output 42 *)
	OUT_CU.tCtr_CustOut[42].Ao		:= OUT_CU.tCtr_Cust42_Out.Y;
	(*scaling parameter watch*)
	Para.rI_Ctr_CustOut_ScalMin[42]	;
	Para.rI_Ctr_CustOut_ScalMax[42]	;

	(* reserve controller output 43 *)
	OUT_CU.tCtr_CustOut[43].Ao		:= OUT_CU.tCtr_Cust43_Out.Y;
	(*scaling parameter watch*)
	Para.rI_Ctr_CustOut_ScalMin[43]	;
	Para.rI_Ctr_CustOut_ScalMax[43]	;

	(* reserve controller output 44 *)
	OUT_CU.tCtr_CustOut[44].Ao		:= OUT_CU.tCtr_Cust44_Out.Y;
	(*scaling parameter watch*)
	Para.rI_Ctr_CustOut_ScalMin[44]	;
	Para.rI_Ctr_CustOut_ScalMax[44]	;

	(* reserve controller output 45 *)
	OUT_CU.tCtr_CustOut[45].Ao		:= OUT_CU.tCtr_Cust45_Out.Y;
	(*scaling parameter watch*)
	Para.rI_Ctr_CustOut_ScalMin[45]	;
	Para.rI_Ctr_CustOut_ScalMax[45]	;

	(*********************************************************************************************************************************)

END_PROGRAM
```

#### c_anaInit.st - Initialisierungscode
```iecst
(********************************************************************
 * COPYRIGHT -- INNIO Company
 ********************************************************************
 * Programm: c_ana
 * Datei: c_anaInit.st
 * Autor: zengeres
 * Erstellt: 30. Januar 2014
 ********************************************************************
 *
 * ALL SETTINGS IN THIS INIT ARE OPTIONAL.
 *
 * If you do not now a special reason, you should NOT SET ANYTHING HERE,
 * since all these settings will be done out of parameter files also.
 *
 ********************************************************************)

PROGRAM _INIT
	(* this parameter defaults will be read only once at first boot, if no Par_CU.dat file exists on the plc*)

	(********************************************)
	(*                                          *)
	(*           ANALOG INPUT SECTION           *)
	(*                                          *)
	(********************************************)

	(*-----------------------------------------------------------------------------*)
	(* Some example lines for intentional disabling of AI warning messages *)
	bBlockW13[03] := FALSE;   (* TRUE will disable Reserve ANALOG IN 1 Warning Signal Error –NUMBER W1177 (rerouted to historical designed message number) *)
	bBlockW13[06] := FALSE;   (* TRUE will disable Reserve ANALOG IN 2 Warning Signal Error –NUMBER W1178 (rerouted to historical designed message number) *)
	bBlockW13[09] := FALSE;   (* TRUE will disable Reserve ANALOG IN 3 Warning Signal Error –NUMBER W1179 (rerouted to historical designed message number) *)
	bBlockW13[12] := FALSE;   (* TRUE will disable Reserve ANALOG IN 4 Warning Signal Error –NUMBER W1180 (rerouted to historical designed message number) *)
	bBlockW13[15] := FALSE;   (* TRUE will disable Reserve ANALOG IN 5 Warning Signal Error –NUMBER W1181 (rerouted to historical designed message number) *)
	bBlockW13[18] := FALSE;   (* TRUE will disable Reserve ANALOG IN 6 Warning Signal Error –NUMBER W1182 (rerouted to historical designed message number) *)
	bBlockW13[21] := FALSE;   (* TRUE will disable Reserve ANALOG IN 7 Warning Signal Error –NUMBER W1183 (rerouted to historical designed message number) *)
	bBlockW13[24] := FALSE;   (* TRUE will disable Reserve ANALOG IN 8 Warning Signal Error –NUMBER W1184 (rerouted to historical designed message number) *)
	(*---*)
	bBlockW13[27] := FALSE;   (* TRUE will disable Reserve ANALOG IN 9 Warning Signal Error –NUMBER W1327*)
	bBlockW13[30] := FALSE;   (* TRUE will disable Reserve ANALOG IN10 Warning Signal Error –NUMBER W1330*)
	bBlockW13[33] := FALSE;   (* TRUE will disable Reserve ANALOG IN11 Warning Signal Error –NUMBER W1333*)
	bBlockW13[36] := FALSE;   (* TRUE will disable Reserve ANALOG IN12 Warning Signal Error –NUMBER W1336*)
	bBlockW13[39] := FALSE;   (* TRUE will disable Reserve ANALOG IN13 Warning Signal Error –NUMBER W1339*)
	bBlockW13[42] := FALSE;   (* TRUE will disable Reserve ANALOG IN14 Warning Signal Error –NUMBER W1342*)
	bBlockW13[45] := FALSE;   (* TRUE will disable Reserve ANALOG IN15 Warning Signal Error –NUMBER W1345*)
	bBlockW13[48] := FALSE;   (* TRUE will disable Reserve ANALOG IN16 Warning Signal Error –NUMBER W1348*)
	(*---*)
	bBlockW13[51] := FALSE;   (* TRUE will disable Reserve ANALOG IN17 Warning Signal Error –NUMBER W1351*)
	bBlockW13[54] := FALSE;   (* TRUE will disable Reserve ANALOG IN18 Warning Signal Error –NUMBER W1354*)
	bBlockW13[57] := FALSE;   (* TRUE will disable Reserve ANALOG IN19 Warning Signal Error –NUMBER W1357*)
	bBlockW13[60] := FALSE;   (* TRUE will disable Reserve ANALOG IN20 Warning Signal Error –NUMBER W1360*)
	bBlockW13[63] := FALSE;   (* TRUE will disable Reserve ANALOG IN21 Warning Signal Error –NUMBER W1363*)
	bBlockW13[66] := FALSE;   (* TRUE will disable Reserve ANALOG IN22 Warning Signal Error –NUMBER W1366*)
	bBlockW13[69] := FALSE;   (* TRUE will disable Reserve ANALOG IN23 Warning Signal Error –NUMBER W1369*)
	bBlockW13[72] := FALSE;   (* TRUE will disable Reserve ANALOG IN24 Warning Signal Error –NUMBER W1372*)
	(*---*)
	bBlockW13[75] := FALSE;   (* TRUE will disable Reserve ANALOG IN25 Warning Signal Error –NUMBER W1375*)
	bBlockW13[78] := FALSE;   (* TRUE will disable Reserve ANALOG IN26 Warning Signal Error –NUMBER W1378*)
	bBlockW13[81] := FALSE;   (* TRUE will disable Reserve ANALOG IN27 Warning Signal Error –NUMBER W1381*)
	bBlockW13[84] := FALSE;   (* TRUE will disable Reserve ANALOG IN28 Warning Signal Error –NUMBER W1384*)
	bBlockW13[87] := FALSE;   (* TRUE will disable Reserve ANALOG IN29 Warning Signal Error –NUMBER W1387*)
	bBlockW13[90] := FALSE;   (* TRUE will disable Reserve ANALOG IN30 Warning Signal Error –NUMBER W1390*)
	bBlockW13[93] := FALSE;   (* TRUE will disable Reserve ANALOG IN31 Warning Signal Error –NUMBER W1393*)
	bBlockW13[96] := FALSE;   (* TRUE will disable Reserve ANALOG IN32 Warning Signal Error –NUMBER W1396*)
	(*---*)
	bBlockW13[99] := FALSE;   (* TRUE will disable Reserve ANALOG IN33 Warning Signal Error –NUMBER W1399*)
	bBlockW14[02] := FALSE;   (* TRUE will disable Reserve ANALOG IN34 Warning Signal Error –NUMBER W1402*)		(*!	 W1400-W1498 USED for Analog In Cannel 34-66 with separate Min and Max and Signalerror Warnings *)
	bBlockW14[05] := FALSE;   (* TRUE will disable Reserve ANALOG IN35 Warning Signal Error –NUMBER W1405*)
	bBlockW14[08] := FALSE;   (* TRUE will disable Reserve ANALOG IN36 Warning Signal Error –NUMBER W1408*)
	bBlockW14[11] := FALSE;   (* TRUE will disable Reserve ANALOG IN37 Warning Signal Error –NUMBER W1411*)
	bBlockW14[14] := FALSE;   (* TRUE will disable Reserve ANALOG IN38 Warning Signal Error –NUMBER W1414*)
	bBlockW14[17] := FALSE;   (* TRUE will disable Reserve ANALOG IN39 Warning Signal Error –NUMBER W1417*)
	bBlockW14[20] := FALSE;   (* TRUE will disable Reserve ANALOG IN40 Warning Signal Error –NUMBER W1420*)
	(*---*)
	bBlockW14[23] := FALSE;   (* TRUE will disable Reserve ANALOG IN41 Warning Signal Error –NUMBER W1423*)
	bBlockW14[26] := FALSE;   (* TRUE will disable Reserve ANALOG IN42 Warning Signal Error –NUMBER W1426*)
	bBlockW14[29] := FALSE;   (* TRUE will disable Reserve ANALOG IN43 Warning Signal Error –NUMBER W1429*)
	bBlockW14[32] := FALSE;   (* TRUE will disable Reserve ANALOG IN44 Warning Signal Error –NUMBER W1432*)
	bBlockW14[35] := FALSE;   (* TRUE will disable Reserve ANALOG IN45 Warning Signal Error –NUMBER W1435*)
	bBlockW14[38] := FALSE;   (* TRUE will disable Reserve ANALOG IN46 Warning Signal Error –NUMBER W1438*)
	bBlockW14[41] := FALSE;   (* TRUE will disable Reserve ANALOG IN47 Warning Signal Error –NUMBER W1441*)
	bBlockW14[44] := FALSE;   (* TRUE will disable Reserve ANALOG IN48 Warning Signal Error –NUMBER W1444*)
	(*---*)
	bBlockW14[47] := FALSE;   (* TRUE will disable Reserve ANALOG IN49 Warning Signal Error –NUMBER W1447*)
	bBlockW14[50] := FALSE;   (* TRUE will disable Reserve ANALOG IN50 Warning Signal Error –NUMBER W1450*)
	bBlockW14[53] := FALSE;   (* TRUE will disable Reserve ANALOG IN51 Warning Signal Error –NUMBER W1453*)
	bBlockW14[56] := FALSE;   (* TRUE will disable Reserve ANALOG IN52 Warning Signal Error –NUMBER W1456*)
	bBlockW14[59] := FALSE;   (* TRUE will disable Reserve ANALOG IN53 Warning Signal Error –NUMBER W1459*)
	bBlockW14[62] := FALSE;   (* TRUE will disable Reserve ANALOG IN54 Warning Signal Error –NUMBER W1462*)
	bBlockW14[65] := FALSE;   (* TRUE will disable Reserve ANALOG IN55 Warning Signal Error –NUMBER W1465*)
	bBlockW14[68] := FALSE;   (* TRUE will disable Reserve ANALOG IN56 Warning Signal Error –NUMBER W1468*)
	(*---*)
	bBlockW14[71] := FALSE;   (* TRUE will disable Reserve ANALOG IN57 Warning Signal Error –NUMBER W1471*)
	bBlockW14[74] := FALSE;   (* TRUE will disable Reserve ANALOG IN58 Warning Signal Error –NUMBER W1474*)
	bBlockW14[77] := FALSE;   (* TRUE will disable Reserve ANALOG IN59 Warning Signal Error –NUMBER W1477*)
	bBlockW14[80] := FALSE;   (* TRUE will disable Reserve ANALOG IN60 Warning Signal Error –NUMBER W1480*)
	(*...continue as needed, if more than 60 AI get activated*)
	(*-----------------------------------------------------------------------------*)

	(* EXAMPLES FOR OPTIONAL HARDCODED CONFIGURATION DEFAULTS:  *)
//	(*Reserve analog input x *)								(* (CONFIGURATION EXAMPLE) *)
//	ParaFactoryDefault.bCustAnaIn_Active[x] :=		FALSE;	(*SET HERE HARDCODED OPTIONALY (runtime changeable)  *)
//	ParaFactoryDefault.rCustAnaIn_ScalMin[x] := 	0.0;	(*SET HERE HARDCODED OPTIONALY (runtime changeable); Active only, when EPLAN definition is set 0-0 *)
//	ParaFactoryDefault.rCustAnaIn_ScalMax[x] := 	1.0;	(*SET HERE HARDCODED OPTIONALY (runtime changeable); Active only, when EPLAN definition is set 0-0 *)
//	ParaFactoryDefault.bCustAnaIn_Set4mA[x] := 		TRUE;	(*OLD, REMOVED*)
//
//	ParaFactoryDefault.iCustAnaIn_MinMaxActive[x] := 3;		(*change customized: 0=no limit messages, 1=activate warning Lo, 2=activate warning hi,  3=activate warning Lo+Hi, (5=activate warning+alarm Lo,  10=activate warning+alarm Hi), 32=alle Störungen und Warnungen EIN   *)
//	ParaFactoryDefault.rCustAnaIn_LimLo[x]	:=		0.1;	(*SET ALARM LIMIT HERE HARDCODED OPTIONALY (runtime changeable)  *)
//	ParaFactoryDefault.rCustAnaIn_LimHi[x]	:=		0.9;	(*set ALARM LIMIT here hardcoded OPTIONALY (runtime changeable)  *)
//	ParaFactoryDefault.rCustAnaIn_Hy[x] := 			0.003; 	(*set hysterese here hardcoded OPTIONALY (runtime changeable)  *)

	(*Reserve analog input 1*)
	ParaFactoryDefault.bCustAnaIn_Active[1] :=		FALSE;
	ParaFactoryDefault.rCustAnaIn_ScalMin[1] := 	0.0;
	ParaFactoryDefault.rCustAnaIn_ScalMax[1] := 	1.0;

	ParaFactoryDefault.iCustAnaIn_MinMaxActive[1] := 3;
	ParaFactoryDefault.rCustAnaIn_LimLo[1]	:=		0.1;
	ParaFactoryDefault.rCustAnaIn_LimHi[1]	:=		0.9;
	ParaFactoryDefault.rCustAnaIn_Hy[1] := 			0.003;

	(*Reserve analog input 2*)
	ParaFactoryDefault.bCustAnaIn_Active[2] :=		FALSE;
	ParaFactoryDefault.rCustAnaIn_ScalMin[2] := 	0.0;
	ParaFactoryDefault.rCustAnaIn_ScalMax[2] := 	1.0;

	ParaFactoryDefault.iCustAnaIn_MinMaxActive[2] := 3;
	ParaFactoryDefault.rCustAnaIn_LimLo[2]	:=		0.1;
	ParaFactoryDefault.rCustAnaIn_LimHi[2]	:=		0.9;
	ParaFactoryDefault.rCustAnaIn_Hy[2] := 			0.003;

	(*Reserve analog input 3*)
	ParaFactoryDefault.bCustAnaIn_Active[3] :=		FALSE;
	ParaFactoryDefault.rCustAnaIn_ScalMin[3] := 	0.0;
	ParaFactoryDefault.rCustAnaIn_ScalMax[3] := 	1.0;

	ParaFactoryDefault.iCustAnaIn_MinMaxActive[3] := 3;
	ParaFactoryDefault.rCustAnaIn_LimLo[3]	:=		0.1;
	ParaFactoryDefault.rCustAnaIn_LimHi[3]	:=		0.9;
	ParaFactoryDefault.rCustAnaIn_Hy[3] := 			0.003;

	(*Reserve analog input 4*)
	ParaFactoryDefault.bCustAnaIn_Active[4]		:= FALSE;

	(* ... *)

	(*Reserve analog input 60*)
	ParaFactoryDefault.bCustAnaIn_Active[60]	:= FALSE;

	(********************************************)
	(*                                          *)
	(*           ANALOG OUTPUT SECTION          *)
	(*                                          *)
	(********************************************)

	(*outputs (only scaling, no activation bit necessary) *)
	ParaFactoryDefault.rCustAnaOut_ScalMax[1] :=	4.0;	(*[mA]; SET HERE HARDCODED OPTIONALY (runtime changeable); Active only, when EPLAN definition is set 0-0 *)
	ParaFactoryDefault.rCustAnaOut_ScalMin[1] :=	20.0;	(*[mA]; SET HERE HARDCODED OPTIONALY (runtime changeable); Active only, when EPLAN definition is set 0-0 *)

	(* ... *)

	(* ...	change or extend this init file customized, if needed.	*)

	(*Check declared array sizze for all AO related types*)  (*iNoOf_AnaOut := 60;*)
	iNoOf_AnaOut_checked[0] := 	iNoOf_AnaOut ;
	iNoOf_AnaOut_checked[1] := SIZEOF(MM2VIS.rCustAnaOut) / SIZEOF(MM2VIS.rCustAnaOut[1]) - 1;									(*Get last element number of declared array*)
	iNoOf_AnaOut_checked[2] := SIZEOF(OUT_CU.tCustAnaOut) / SIZEOF(OUT_CU.tCustAnaOut[1]) - 1;				(*Get last element number of declared array*)
	iNoOf_AnaOut_checked[3] := SIZEOF(Para.rCustAnaOut_ScalMin) / SIZEOF(Para.rCustAnaOut_ScalMin[1]) - 1;	(*Get last element number of declared array*)
	iNoOf_AnaOut_checked[4] := SIZEOF(Para.rCustAnaOut_ScalMax) / SIZEOF(Para.rCustAnaOut_ScalMax[1]) - 1;	(*Get last element number of declared array*)
	iNoOf_AnaOut_checked[5] := SIZEOF(Para.bCustAnaOut_Active) / SIZEOF(Para.bCustAnaOut_Active[1]) - 1;		(*Get last element number of declared array*)
	iNoOf_AnaOut_checked[6] := SIZEOF(Para.rI_CustAnaOut_ScalMin) / SIZEOF(Para.rI_CustAnaOut_ScalMin[1]) - 1;	(*Get last element number of declared array*)
	iNoOf_AnaOut_checked[7] := SIZEOF(Para.rI_CustAnaOut_ScalMax) / SIZEOF(Para.rI_CustAnaOut_ScalMax[1]) - 1;	(*Get last element number of declared array*)
	FOR i := 1 TO 7 DO
		iNoOf_AnaOut_checked[0] := MIN(iNoOf_AnaOut_checked[0] , iNoOf_AnaOut_checked[i] );
	END_FOR
	bErr_NoOf_AnaOut := iNoOf_AnaOut <> iNoOf_AnaOut_checked[0] ;

	(********************************************)
	(*                                          *)
	(*         CONTROLLER OUTPUT SECTION        *)
	(*                                          *)
	(********************************************)

	(*controller outputs (only scaling, no activation bit necessary) *)
	ParaFactoryDefault.rCtr_CustOut_ScalMax[1] :=	4.0;	(*[mA]; SET HERE HARDCODED OPTIONALY (runtime changeable); Active only, when EPLAN definition is set 0-0 *)
	ParaFactoryDefault.rCtr_CustOut_ScalMin[1] :=	20.0;	(*[mA]; SET HERE HARDCODED OPTIONALY (runtime changeable); Active only, when EPLAN definition is set 0-0 *)

	(* ... *)

	(* ...	change or extend this init file customized, if needed.	*)

(********************** no changes bejond this line ****************************)

(*******************************************************************************)
(*   Compatibility code section below. NO NEED TO CHANGE on new XT4 engines!   *)
(*******************************************************************************)																			rReplaceMeWithLocaleVarName;		(* this statements mark places all over the code, that shoud be edited according to customer needs, but PLEASE leaf this occurence here unchanged for internal purposes*)
	(**OLD**)
	(*Old extension for analog inputs: Signal-Typ *)
	ParaFactoryDefault.iCustAnaIn_Typ[1] ; //:= 15;	 		(*(PARTLY OBSOLETE). ONLY USED TO ACTIVATE AN ADDITIONAL SCALING (without HAL changes) or for COMPATIBILITY WITH OLD XT and XT3 ENGINES *)
	(*0 ... mA oder +V	1 ... Pt100	2 ... NiCr-Ni	4 ... 4mA to 20mA  	(OBSOLETE TYPE CODES, numbers below 10 are here stated only for compatibility)
	Additional Scaling:	10... mA oder +V to paravalues scaled	15... Normed to paravalues scaled?		16...paravalues scaled to Normed?*)

	(*Old extension for analog inputs: physical unit display code for VIS  *)
	ParaFactoryDefault.iCustAnaIn_Unit[1];	// := 0;		(*OBSOLETE. _Unit parameter is ONLY STATED HERE FOR COMPATIBILITY WITH OLD XT and XT3 ENGINES. Do not use on new engines.*)
	(*	1  = °C		2  = bar		3  = mbar	4  = kW		5  = kVAr		6  = mV		7  = V			8  = mA		9  = A			10 = kWh
	11 = MWh	12 = 0,1 MWh	13 = kVArh	14 = MVArh	15 = 0,1 MVArh	16 = m3		17 = 1000 m3	18 = Nm3	19 = 1000 Nm3	20 = m3/h
	21 = Nm3/h	22 = %			23 = 1/min	24 = Hz		25 = s			26 = h		27 = l			28 = °F		29 = psi		30 = mpsi	0  = none	*)
	(**/OLD**)

END_PROGRAM
```

#### c_ana.var - Lokale Variablen
```iecst
VAR
	rReplaceMeWithLocaleVarName : REAL;
END_VAR
VAR CONSTANT
	rConnectYourVariableHere : REAL := 0.0; (*replace this tag with your variable*)
END_VAR
VAR
	iCnt_AnaOut : INT := 0;
	iNoOf_AnaOut_checked : ARRAY[0..9] OF INT := [10(0)]; (*Check realy declared array sizze*)
	i : INT := 0;
END_VAR
```

### Program Logical/Customized/c_scal (IEC, version 4.11.0) - Scaling Blocks for internal use

#### c_scalCyclic.st - Cyclic code
```iecst
(*******************************************************************************
CUSTOMIZED: c_scal 		reserve scaling blocks (cyclic)

This code is confidential AND proprietary to the INNIO Company.
It may NOT be used in any form, or reproduced in any manner,
without written permission of the INNIO Company.
Copyright, INNIO Company, 2022

Customized modifications: -
------------------------

History:
-------
V4.00	29.09.2021	Heim Markus	generated, new
V4.11.0	07.12.2021	Zengerer	integrate initial version

Instructions FOR use:
--------------------
-
Outstandings:
------------

*******************************************************************************)

PROGRAM _CYCLIC

	(* customizable scaling block n
	*Input*
	IN_CU.rScalBlock_X[n]			:=	rReplaceMeWithVarname; 				* input variable TO get scaling
	*Parameter*
	xScalBlock[n].Type				:=	Para.iCust_ScalingBlock_Typ[n];		* 0 = deactivated | 1 = scaling with limits | 2 = scaling without limits
	xScalBlock[n].X1				:=	Para.rCust_ScalingBlock_X1[n];		* change to scaling parameter; initial default value is 0.0
	xScalBlock[n].X2				:=	Para.rCust_ScalingBlock_X2[n];		* change to scaling parameter; initial default value is 1.0
	xScalBlock[n].Y1				:=	Para.rCust_ScalingBlock_Y1[n];		* change to scaling parameter; initial default value is 0.0
	xScalBlock[n].Y2				:=	Para.rCust_ScalingBlock_Y2[n];		* change to scaling parameter; initial default value is 1.0
	*Visu*
	MM2VIS.rCustScalingBlock_X[n]	:=	xScalBlock[n].X;					* Visu
	MM2VIS.rCustScalingBlock_Y[n]	:=	xScalBlock[n].Y;					* Visu
	*Output*
	rReplaceMeWithVarname			:=	xScalBlock[n].Y;					* optional scaled output variable connector
	bReplaceMeWithVarname			:=	xScalBlock[n].Err;					* optional error Flag connector; connect alarm messaging only if need occures

	(*******************************************************************************************************************************)
	(* customizable scaling block 1*)
	(*Input*)
	IN_CU.rScalBlock_X[1];											(* connect input variable here *)
	(*Output*)
	rReplaceMeWithVarname			:=	OUT_CU.rScalBlock_Y[1];		(* option to connect output variable here *)
	bReplaceMeWithVarname			:=	OUT_CU.bScalBlock_Err[1];	(* connect optional error Flag if needed *)

	(*******************************************************************************************************************************)
	(* customizable scaling block 2*)
	(*Input*)
	IN_CU.rScalBlock_X[2];											(* connect input variable here *)
	(*Output*)
	rReplaceMeWithVarname			:=	OUT_CU.rScalBlock_Y[2];
	bReplaceMeWithVarname			:=	OUT_CU.bScalBlock_Err[2];

	(*******************************************************************************************************************************)
	(* customizable scaling block 3*)
	(*Input*)
	IN_CU.rScalBlock_X[3];											(* connect input variable here *)
	(*Output*)
	rReplaceMeWithVarname			:=	OUT_CU.rScalBlock_Y[3];
	bReplaceMeWithVarname			:=	OUT_CU.bScalBlock_Err[3];

	(*******************************************************************************************************************************)
	(* customizable scaling block 4*)
	(*Input*)
	IN_CU.rScalBlock_X[4];											(* connect input variable here *)
	(*Output*)
	rReplaceMeWithVarname			:=	OUT_CU.rScalBlock_Y[4];
	bReplaceMeWithVarname			:=	OUT_CU.bScalBlock_Err[4];

	(*******************************************************************************************************************************)
	(* customizable scaling block 5*)
	(*Input*)
	IN_CU.rScalBlock_X[5];											(* connect input variable here *)
	(*Output*)
	rReplaceMeWithVarname			:=	OUT_CU.rScalBlock_Y[5];
	bReplaceMeWithVarname			:=	OUT_CU.bScalBlock_Err[5];

	(*******************************************************************************************************************************)
	(* customizable scaling block 6*)
	(*Input*)
	IN_CU.rScalBlock_X[6];											(* connect input variable here *)
	(*Output*)
	rReplaceMeWithVarname			:=	OUT_CU.rScalBlock_Y[6];
	bReplaceMeWithVarname			:=	OUT_CU.bScalBlock_Err[6];

	(*******************************************************************************************************************************)
	(* customizable scaling block 7*)
	(*Input*)
	IN_CU.rScalBlock_X[7];											(* connect input variable here *)
	(*Output*)
	rReplaceMeWithVarname			:=	OUT_CU.rScalBlock_Y[7];
	bReplaceMeWithVarname			:=	OUT_CU.bScalBlock_Err[7];

	(*******************************************************************************************************************************)
	(* customizable scaling block 8*)
	(*Input*)
	IN_CU.rScalBlock_X[8];											(* connect input variable here *)
	(*Output*)
	rReplaceMeWithVarname			:=	OUT_CU.rScalBlock_Y[8];
	bReplaceMeWithVarname			:=	OUT_CU.bScalBlock_Err[8];

	(*******************************************************************************************************************************)
	(* customizable scaling block 9*)
	(*Input*)
	IN_CU.rScalBlock_X[9];											(* connect input variable here *)
	(*Output*)
	rReplaceMeWithVarname			:=	OUT_CU.rScalBlock_Y[9];
	bReplaceMeWithVarname			:=	OUT_CU.bScalBlock_Err[9];

	(*******************************************************************************************************************************)
	(* customizable scaling block 10*)
	(*Input*)
	IN_CU.rScalBlock_X[10];											(* connect input variable here *)
	(*Output*)
	rReplaceMeWithVarname			:=	OUT_CU.rScalBlock_Y[10];
	bReplaceMeWithVarname			:=	OUT_CU.bScalBlock_Err[10];

	(*** DEFAULT CONFIG END ********************************************************************************************************)
	(*** DEFAULT CONFIG END  - ADD VIS EXTENTION PACKAGE to use more than the default number of channels ***************************)
	(*** DEFAULT CONFIG END ********************************************************************************************************)

	(*******************************************************************************************************************************)
	(* customizable scaling block 11*)
	(*Input*)
	IN_CU.rScalBlock_X[11];											(* connect input variable here *)
	(*Output*)
	rReplaceMeWithVarname			:=	OUT_CU.rScalBlock_Y[11];
	bReplaceMeWithVarname			:=	OUT_CU.bScalBlock_Err[11];

	(*******************************************************************************************************************************)
	(* customizable scaling block 12*)
	(*Input*)
	IN_CU.rScalBlock_X[12];											(* connect input variable here *)
	(*Output*)
	rReplaceMeWithVarname			:=	OUT_CU.rScalBlock_Y[12];
	bReplaceMeWithVarname			:=	OUT_CU.bScalBlock_Err[12];

	(*******************************************************************************************************************************)
	(* customizable scaling block 13*)
	(*Input*)
	IN_CU.rScalBlock_X[13];											(* connect input variable here *)
	(*Output*)
	rReplaceMeWithVarname			:=	OUT_CU.rScalBlock_Y[13];
	bReplaceMeWithVarname			:=	OUT_CU.bScalBlock_Err[13];

	(*******************************************************************************************************************************)
	(* customizable scaling block 14*)
	(*Input*)
	IN_CU.rScalBlock_X[14];											(* connect input variable here *)
	(*Output*)
	rReplaceMeWithVarname			:=	OUT_CU.rScalBlock_Y[14];
	bReplaceMeWithVarname			:=	OUT_CU.bScalBlock_Err[14];

	(*******************************************************************************************************************************)
	(* customizable scaling block 15*)
	(*Input*)
	IN_CU.rScalBlock_X[15];											(* connect input variable here *)
	(*Output*)
	rReplaceMeWithVarname			:=	OUT_CU.rScalBlock_Y[15];
	bReplaceMeWithVarname			:=	OUT_CU.bScalBlock_Err[15];

	(*******************************************************************************************************************************)
	(* customizable scaling block 16*)
	(*Input*)
	IN_CU.rScalBlock_X[16];											(* connect input variable here *)
	(*Output*)
	rReplaceMeWithVarname			:=	OUT_CU.rScalBlock_Y[16];
	bReplaceMeWithVarname			:=	OUT_CU.bScalBlock_Err[16];

	(*******************************************************************************************************************************)
	(* customizable scaling block 17*)
	(*Input*)
	IN_CU.rScalBlock_X[17];											(* connect input variable here *)
	(*Output*)
	rReplaceMeWithVarname			:=	OUT_CU.rScalBlock_Y[17];
	bReplaceMeWithVarname			:=	OUT_CU.bScalBlock_Err[17];

	(*******************************************************************************************************************************)
	(* customizable scaling block 18*)
	(*Input*)
	IN_CU.rScalBlock_X[18];											(* connect input variable here *)
	(*Output*)
	rReplaceMeWithVarname			:=	OUT_CU.rScalBlock_Y[18];
	bReplaceMeWithVarname			:=	OUT_CU.bScalBlock_Err[18];

	(*******************************************************************************************************************************)
	(* customizable scaling block 19*)
	(*Input*)
	IN_CU.rScalBlock_X[19];											(* connect input variable here *)
	(*Output*)
	rReplaceMeWithVarname			:=	OUT_CU.rScalBlock_Y[19];
	bReplaceMeWithVarname			:=	OUT_CU.bScalBlock_Err[19];

	(*******************************************************************************************************************************)
	(* customizable scaling block 20*)
	(*Input*)
	IN_CU.rScalBlock_X[20];											(* connect input variable here *)
	(*Output*)
	rReplaceMeWithVarname			:=	OUT_CU.rScalBlock_Y[20];
	bReplaceMeWithVarname			:=	OUT_CU.bScalBlock_Err[20];

	(*******************************************************************************************************************************)
	(* customizable scaling block 21*)
	(*Input*)
	IN_CU.rScalBlock_X[21];											(* connect input variable here *)
	(*Output*)
	rReplaceMeWithVarname			:=	OUT_CU.rScalBlock_Y[21];
	bReplaceMeWithVarname			:=	OUT_CU.bScalBlock_Err[21];

	(*******************************************************************************************************************************)
	(* customizable scaling block 22*)
	(*Input*)
	IN_CU.rScalBlock_X[22];											(* connect input variable here *)
	(*Output*)
	rReplaceMeWithVarname			:=	OUT_CU.rScalBlock_Y[22];
	bReplaceMeWithVarname			:=	OUT_CU.bScalBlock_Err[22];

	(*******************************************************************************************************************************)
	(* customizable scaling block 23*)
	(*Input*)
	IN_CU.rScalBlock_X[23];											(* connect input variable here *)
	(*Output*)
	rReplaceMeWithVarname			:=	OUT_CU.rScalBlock_Y[23];
	bReplaceMeWithVarname			:=	OUT_CU.bScalBlock_Err[23];

	(*******************************************************************************************************************************)
	(* customizable scaling block 24*)
	(*Input*)
	IN_CU.rScalBlock_X[24];											(* connect input variable here *)
	(*Output*)
	rReplaceMeWithVarname			:=	OUT_CU.rScalBlock_Y[24];
	bReplaceMeWithVarname			:=	OUT_CU.bScalBlock_Err[24];

	(*******************************************************************************************************************************)
	(* customizable scaling block 25*)
	(*Input*)
	IN_CU.rScalBlock_X[25];											(* connect input variable here *)
	(*Output*)
	rReplaceMeWithVarname			:=	OUT_CU.rScalBlock_Y[25];
	bReplaceMeWithVarname			:=	OUT_CU.bScalBlock_Err[25];

	(*******************************************************************************************************************************)
	(* customizable scaling block 26*)
	(*Input*)
	IN_CU.rScalBlock_X[26];											(* connect input variable here *)
	(*Output*)
	rReplaceMeWithVarname			:=	OUT_CU.rScalBlock_Y[26];
	bReplaceMeWithVarname			:=	OUT_CU.bScalBlock_Err[26];

	(*******************************************************************************************************************************)
	(* customizable scaling block 27*)
	(*Input*)
	IN_CU.rScalBlock_X[27];											(* connect input variable here *)
	(*Output*)
	rReplaceMeWithVarname			:=	OUT_CU.rScalBlock_Y[27];
	bReplaceMeWithVarname			:=	OUT_CU.bScalBlock_Err[27];

	(*******************************************************************************************************************************)
	(* customizable scaling block 28*)
	(*Input*)
	IN_CU.rScalBlock_X[28];											(* connect input variable here *)
	(*Output*)
	rReplaceMeWithVarname			:=	OUT_CU.rScalBlock_Y[28];
	bReplaceMeWithVarname			:=	OUT_CU.bScalBlock_Err[28];

	(*******************************************************************************************************************************)
	(* customizable scaling block 29*)
	(*Input*)
	IN_CU.rScalBlock_X[29];											(* connect input variable here *)
	(*Output*)
	rReplaceMeWithVarname			:=	OUT_CU.rScalBlock_Y[29];
	bReplaceMeWithVarname			:=	OUT_CU.bScalBlock_Err[29];

	(*******************************************************************************************************************************)
	(* customizable scaling block 30*)
	(*Input*)
	IN_CU.rScalBlock_X[30];											(* connect input variable here *)
	(*Output*)
	rReplaceMeWithVarname			:=	OUT_CU.rScalBlock_Y[30];
	bReplaceMeWithVarname			:=	OUT_CU.bScalBlock_Err[30];

	(*******************************************************************************************************************************)
	(*	END OF CONFIGURATION AREA; no changes necessary below this line *)
	(******************************************************************************************************************************)
	(*parameter assignment and function call for scaling blocks*)
	FOR n := 1 TO 30 BY 1 DO
		(*Parameter*)
		xScalBlock[n].Type			:=	Para.iCust_ScalingBlock_Typ[n];		(* 0 = deactivated | 1 = scaling with limits | 2 = scaling without limits *)
		xScalBlock[n].X				:=	IN_CU.rScalBlock_X[n];				(* input variable connector *)
		xScalBlock[n].X1			:=	Para.rCust_ScalingBlock_X1[n];
		xScalBlock[n].X2			:=	Para.rCust_ScalingBlock_X2[n];
		xScalBlock[n].Y1			:=	Para.rCust_ScalingBlock_Y1[n];
		xScalBlock[n].Y2			:=	Para.rCust_ScalingBlock_Y2[n];
		xScalBlock[n]();	(*function call*)
		(*Output*)
		OUT_CU.rScalBlock_Y[n]		:=	xScalBlock[n].Y;					(* output variable connector *)
		OUT_CU.bScalBlock_Err[n]	:=	xScalBlock[n].Err;					(* optional error Flag connector, if needed *)
		(*Visu*)
		MM2VIS.rCustScalingBlock_X[n]	:=	xScalBlock[n].X;
		MM2VIS.rCustScalingBlock_Y[n]	:=	xScalBlock[n].Y;
	END_FOR

END_PROGRAM
```

#### c_scalInit.st - Initialization code
```iecst
(*******************************************************************************
CUSTOMIZED: c_scal 		reserve scaling blocks (init)

This code is confidential AND proprietary to the INNIO Company.
It may NOT be used in any form, or reproduced in any manner,
without written permission of the INNIO Company.
Copyright, INNIO Company, 2022

Customized modifications: -
------------------------

History:
-------
V4.00	29.09.2021	Heim Markus generated, new
V4.11.0	07.12.2021	Zengerer	integrate initial version, ParaFactoryDefault

Instructions for use:
--------------------
-
Outstandings:
------------
-

*******************************************************************************)

PROGRAM _INIT

	(*initial Type = 0*)
	FOR n := 1 TO 30 BY 1 DO
		xScalBlock[n].Type := 0;

		ParaFactoryDefault.rCust_ScalingBlock_X2[n] := 1.0;		(* default before first parameter load *)
		ParaFactoryDefault.rCust_ScalingBlock_Y2[n] := 1.0; 	(* default before first parameter load *)
	END_FOR

END_PROGRAM
```

#### c_scal.var - Local variables
```iecst
(********************************************************************
 * COPYRIGHT -- INNIO Company
 ********************************************************************
 * Program: c_scal
 * File: c_scal.var
 * Author: Heim Markus
 * Created: 29.09.2021
 ********************************************************************
 * Local variables of program c_scal
 ********************************************************************)
VAR
	rReplaceMeWithVarname : REAL; (*void*)
	bReplaceMeWithVarname : BOOL; (*void*)
	xScalBlock : ARRAY[0..30] OF ScalBlock := [31((0))]; (*custom scaling Blocks array*)
	n : USINT := 0; (*Scaling Blocks internal counter*)
END_VAR
```

#### ScalBlock.fun - Exported functions and function blocks
```iecst
FUNCTION_BLOCK ScalBlock
	VAR_INPUT
		Type : INT; (*Type of scaling*)
		X : REAL; (*X input value*)
		X1 : REAL; (*X1 input Parameter*)
		X2 : REAL; (*X2 input Parameter*)
		Y1 : REAL; (*Y1 input Parameter*)
		Y2 : REAL; (*Y2 input Parameter*)
	END_VAR
	VAR_OUTPUT
		Y : REAL; (*Y output value*)
		Err : BOOL; (*Error Flag*)
	END_VAR
	VAR
		xLCRLimScal : LCRLimScal; (*scaling with limitation*)
		xLCRScal : LCRScal; (*scaling without limitation*)
	END_VAR
END_FUNCTION_BLOCK
```

#### ScalBlock.st - function scaling blocks
```iecst
(********************************************************************
This code is confidential AND proprietary to the INNIO Company.
It may NOT be used in any form, or reproduced in any manner, without the express
written permission of the INNIO Company.
Copyright, INNIO Company, 2022

Customized modifications: -
------------------------

History:
-------
V4.11.00	29.09.2021	Heim Markus	created Scaling Bock FUB

Instructions FOR use:
--------------------

Outstandings: -
------------
*******************************************************************************)

FUNCTION_BLOCK ScalBlock

	IF 		Type = 0 THEN  		(* 0 = deactivated *)
		Y	:=	0.0;
	ELSIF	Type = 1 THEN		(* 1 = scaling with limits *)
		IF X1 = X2 THEN			(*Error Flag with X1 = X2*)
			Err :=	TRUE;
			Y   := 0.0;
		ELSE
			xLCRLimScal.x	:=	X;
			xLCRLimScal.x1	:=	X1;
			xLCRLimScal.x2	:=	X2;
			xLCRLimScal.y1	:=	Y1;
			xLCRLimScal.y2	:=	Y2;
			xLCRLimScal();
			Y	:=	xLCRLimScal.y;
		END_IF
	ELSIF	Type = 2 THEN		(* 2 = scaling without limits *)
		IF X1 = X2 THEN			(*Error Flag with X1 = X2*)
			Err :=	TRUE;
			Y   := 0.0;
		ELSE
			xLCRScal.x		:=	X;
			xLCRScal.x1		:=	X1;
			xLCRScal.x2		:=	X2;
			xLCRScal.y1		:=	Y1;
			xLCRScal.y2		:=	Y2;
			xLCRScal();
			Y	:=	xLCRScal.y;
		END_IF
	ELSIF	Type = 3 THEN		(* 3 = Y value = X value *)
		Y	:=	X;
	ELSE
		Err :=	TRUE; 			(*Error Flag with undefined stat*)
		Y   := 0.0;
	END_IF

END_FUNCTION_BLOCK
```

### Program Logical/Customized/c_par (IEC, version 4.04.0) - Handling of prepared customizable parameter values
